(* CODESYS project skyWell.v2.01.project

Project tree, tasks and I/O mapping:
  Device : CODESYS SoftMotion RTE V3, 3S - Smart Software Solutions GmbH, order no. 309015, version 3.5.9.50
    application Application
      libraries: Standard, * (System); VisuDialogs, * (System); SysTime, 3.5.9.0 (System); SysFile, 3.5.9.0 (System); SysStr23, 3.5.8.0 (System); CAA DTUtil Extern, 3.5.10.0 (CAA Technical Workgroup); AC_Persistence, 3.5.10.0 (3S - Smart Software Solutions GmbH); modbus tcp serverAndClient, 1.0.1 (深圳人通长沙研究院); TCP, 3.5.9.50 (3S - Smart Software Solutions GmbH); SysDir, 3.5.8.0 (System); SysTime23, 3.5.2.0 (System); CAA File, 3.5.9.0 (CAA Technical Workgroup)
      task ceilingRail (cyclic, interval t#20ms, priority 1) calls ceilingRailAct
      task healthyData1 (cyclic, interval t#500ms, priority 1) calls tcpUploader
      task VISU_TASK (cyclic, interval 100 ms, priority 31) calls VisuElems.Visu_Prg
      task canSend (cyclic, interval t#20ms, priority 1) calls canTx
      task modbus (cyclic, interval t#20ms, priority 1) calls modbusAct
      task canReceive (cyclic, interval 4 ms, priority 0) calls canRx
      task healthyData2 (cyclic, interval t#10ms, priority 1) calls fileSaver
      rail_ceiling/
        struct_ceiling_rail/
          data type propValveModule_Ti
          data type PropValveTiX
          data type UICell_OilBlock_Ti
        program ceilingRailAct [ST]: initName, statusDisplayTi, initRange, statusPercentCalcTi, cmdDeliverTi, cmdDeliverPlate, cmdDeliverManual
        function cmdExecuteT [ST]
        program positionRecord [ST]
      can/
        structCan/
          data type Can_baseframe
          data type Can_BUS_8Inputs
          data type Can_BUS_8Outputs
          data type Can_Bus_RXMsg_Buff
          data type Can_Bus_TXMsg_Buff
        function CAN_Send_Data_SWMC [ST]
        function swmc_C05_Rx [ST]
        function swmc_C05_Tx [ST]
        function swmc_C06_Tx [ST]
        function swmc_C12_Rx [ST]
        function CAN_Read_Data_SWMC [ST]
        program canTx [ST]
        program canRx [ST]
        function swmc_C06_Rx [ST]
      global variables gImple
      global variables gUI
      global variables gCan
      display/
        Module/
          visualisation OilBlock_PrimButton
          visualisation OilBlock_PrimInfo
          visualisation ModuleX2
          visualisation ModuleX1
          visualisation ModuleX3
          visualisation ModuleX8
          visualisation ModuleX4
          visualisation ModuleX5
          visualisation ModuleDTD
        OrigTi/
          visualisation Ceiling_Rail2
          visualisation Ceiling_Rail1
          visualisation Ceiling_Rail_345
          visualisation Ceiling_Rail6
          visualisation Ceiling_Rail7
          visualisation Ceiling_Rail_12
          visualisation Ceiling_Rail_67
          visualisation Ceiling_Rail_Plate
          visualisation ManualMode
        visualisation Ceiling_Rail
      public_datum/
        yy_station/
          struct_yystation/
            data type YyStation_Cmd
            data type YyStation_Status
            data type YyStation
        oilblock/
          struct/
            data type OilBlockUnit_Base
            data type OilBlockUnit_Status
            data type OilBlockUnit_Cmdx
            data type OilBlockUnit_Status_Loc
            data type OilBlockUnit_Status_PosVal
            data type UICell_OilBlock_Module
            data type UICell_OilBlock_Module_Info
            data type UICell_OilBlock_Module_Button
            data type UICell_OilBlock_Tag
            data type OilBlockUnit_RangeRec
            data type OilBlockUnit_Add
            data type UICell_ManualMode
            data type UICell_OilBlockPlat_Module
        cmdcheck/
          function block checkoilUnit [ST]
          function GetPositionValueOfUnit8 [ST]
          data type cmdStat
          function block checkoilGropisDoneX8 [ST]
          function fGetUnitStat [ST]
          function block percentCalc [ST]
          function block syncUnitCheck [ST]
          function fUICmdDetect [ST]
        datarecord/
          function block datSave [ST]
          function block logSave [ST]
      global variables gModbus
      modbus/
        struct_modbus/
          data type ModbusStructx
          data type Modbus_Commandx
          data type Modbus_Statusx
          data type Modbus_Heartbeatx
          data type Modbus_ActionIndex
        program modbusAct [ST]: initAddrPacket, handleToken, handleCommand1, handleStatus1, executeCmd, getStatus
        function block getObjIndexC [ST]
        function block getObjIndexE [ST]
        function block getObjIndexR [ST]
        function block getColumnStr [ST]
      rail_plate/
        function cmdExecutePlate [ST]
        data type plateCmd
        data type plateStat
      dataUpload/
        function block tcpUpload [ST]: send
        function block findMasterCtrl [ST]
        function block getStateByIdx [ST]
        program tcpUploader [ST]: prepareMetaData
        function block fileSave [ST]: new, close, write, createDir
        program fileSaver [ST]: getData
    SoftMotion General Axis Pool
    EtherCAT_Master : EtherCAT Master, 3S - Smart Software Solutions GmbH, version 3.5.10.0
        settings: NetworkName = '本地连接 2'; NetworkName = "本地连接 2"; SelectNetworkByName = False; SrcAddress1 = 26861; SrcAddress2 = 2752489275
      EK1100_0030_2 : EK1100-0030 EtherCAT Coupler (2A E-Bus, 4kV galv. iso.), Beckhoff Automation GmbH & Co. KG, order no. EK1100-0030, version Revision=16#0011001E
          settings: DC sync0 cycletime = 4000; DC sync1 cycletime = 4000
        EL6751_CANMiniDriver_1 : EL6751 CAN MiniDriver (8 Messages), Beckhoff Automation GmbH, version 3.5.9.0
            settings: DC sync0 cycletime = 4000; DC sync1 cycletime = 4000
            unmapped channels: TxCounter, RxCounter, NoOfTxMessages, TxMsg1_TransactionNumber, TxMsg1_CobId, TxMsg1_Byte1, TxMsg1_Byte2, TxMsg1_Byte3, TxMsg1_Byte4, TxMsg1_Byte5, TxMsg1_Byte6, TxMsg1_Byte7, TxMsg1_Byte8, TxMsg2_TransactionNumber, TxMsg2_CobId, TxMsg2_Byte1, TxMsg2_Byte2, TxMsg2_Byte3, TxMsg2_Byte4, TxMsg2_Byte5, TxMsg2_Byte6, TxMsg2_Byte7, TxMsg2_Byte8, TxMsg3_TransactionNumber, TxMsg3_CobId, TxMsg3_Byte1, TxMsg3_Byte2, TxMsg3_Byte3, TxMsg3_Byte4, TxMsg3_Byte5, TxMsg3_Byte6, TxMsg3_Byte7, TxMsg3_Byte8, TxMsg4_TransactionNumber, TxMsg4_CobId, TxMsg4_Byte1, TxMsg4_Byte2, TxMsg4_Byte3, TxMsg4_Byte4, TxMsg4_Byte5,
              TxMsg4_Byte6, TxMsg4_Byte7, TxMsg4_Byte8, TxMsg5_TransactionNumber, TxMsg5_CobId, TxMsg5_Byte1, TxMsg5_Byte2, TxMsg5_Byte3, TxMsg5_Byte4, TxMsg5_Byte5, TxMsg5_Byte6, TxMsg5_Byte7, TxMsg5_Byte8, TxMsg6_TransactionNumber, TxMsg6_CobId, TxMsg6_Byte1, TxMsg6_Byte2, TxMsg6_Byte3, TxMsg6_Byte4, TxMsg6_Byte5, TxMsg6_Byte6, TxMsg6_Byte7, TxMsg6_Byte8, TxMsg7_TransactionNumber, TxMsg7_CobId, TxMsg7_Byte1, TxMsg7_Byte2, TxMsg7_Byte3, TxMsg7_Byte4, TxMsg7_Byte5, TxMsg7_Byte6, TxMsg7_Byte7, TxMsg7_Byte8, TxMsg8_TransactionNumber, TxMsg8_CobId, TxMsg8_Byte1, TxMsg8_Byte2, TxMsg8_Byte3, TxMsg8_Byte4, TxMsg8_Byte5,
              TxMsg8_Byte6, TxMsg8_Byte7, TxMsg8_Byte8, CAN Control, TxCounter, RxCounter, NoOfRxMessages, TransactionNumber, RxMsg1_CobId, RxMsg1_Byte1, RxMsg1_Byte2, RxMsg1_Byte3, RxMsg1_Byte4, RxMsg1_Byte5, RxMsg1_Byte6, RxMsg1_Byte7, RxMsg1_Byte8, RxMsg2_CobId, RxMsg2_Byte1, RxMsg2_Byte2, RxMsg2_Byte3, RxMsg2_Byte4, RxMsg2_Byte5, RxMsg2_Byte6, RxMsg2_Byte7, RxMsg2_Byte8, RxMsg3_CobId, RxMsg3_Byte1, RxMsg3_Byte2, RxMsg3_Byte3, RxMsg3_Byte4, RxMsg3_Byte5, RxMsg3_Byte6, RxMsg3_Byte7, RxMsg3_Byte8, RxMsg4_CobId, RxMsg4_Byte1, RxMsg4_Byte2, RxMsg4_Byte3, RxMsg4_Byte4,
              RxMsg4_Byte5, RxMsg4_Byte6, RxMsg4_Byte7, RxMsg4_Byte8, RxMsg5_CobId, RxMsg5_Byte1, RxMsg5_Byte2, RxMsg5_Byte3, RxMsg5_Byte4, RxMsg5_Byte5, RxMsg5_Byte6, RxMsg5_Byte7, RxMsg5_Byte8, RxMsg6_CobId, RxMsg6_Byte1, RxMsg6_Byte2, RxMsg6_Byte3, RxMsg6_Byte4, RxMsg6_Byte5, RxMsg6_Byte6, RxMsg6_Byte7, RxMsg6_Byte8, RxMsg7_CobId, RxMsg7_Byte1, RxMsg7_Byte2, RxMsg7_Byte3, RxMsg7_Byte4, RxMsg7_Byte5, RxMsg7_Byte6, RxMsg7_Byte7, RxMsg7_Byte8, RxMsg8_CobId, RxMsg8_Byte1, RxMsg8_Byte2, RxMsg8_Byte3, RxMsg8_Byte4, RxMsg8_Byte5, RxMsg8_Byte6, RxMsg8_Byte7, RxMsg8_Byte8,
              CAN State, Align, RX Error Counter, TX Error Counter
          CANbus
              settings: NetID = 2
      EK1100_0030_1 : EK1100-0030 EtherCAT Coupler (2A E-Bus, 4kV galv. iso.), Beckhoff Automation GmbH & Co. KG, order no. EK1100-0030, version Revision=16#0011001E
          settings: DC sync0 cycletime = 4000; DC sync1 cycletime = 4000
        EL6751_CANMiniDriver : EL6751 CAN MiniDriver (8 Messages), Beckhoff Automation GmbH, version 3.5.9.0
            settings: DC sync0 cycletime = 4000; DC sync1 cycletime = 4000
            unmapped channels: TxCounter, RxCounter, NoOfTxMessages, TxMsg1_TransactionNumber, TxMsg1_CobId, TxMsg1_Byte1, TxMsg1_Byte2, TxMsg1_Byte3, TxMsg1_Byte4, TxMsg1_Byte5, TxMsg1_Byte6, TxMsg1_Byte7, TxMsg1_Byte8, TxMsg2_TransactionNumber, TxMsg2_CobId, TxMsg2_Byte1, TxMsg2_Byte2, TxMsg2_Byte3, TxMsg2_Byte4, TxMsg2_Byte5, TxMsg2_Byte6, TxMsg2_Byte7, TxMsg2_Byte8, TxMsg3_TransactionNumber, TxMsg3_CobId, TxMsg3_Byte1, TxMsg3_Byte2, TxMsg3_Byte3, TxMsg3_Byte4, TxMsg3_Byte5, TxMsg3_Byte6, TxMsg3_Byte7, TxMsg3_Byte8, TxMsg4_TransactionNumber, TxMsg4_CobId, TxMsg4_Byte1, TxMsg4_Byte2, TxMsg4_Byte3, TxMsg4_Byte4, TxMsg4_Byte5,
              TxMsg4_Byte6, TxMsg4_Byte7, TxMsg4_Byte8, TxMsg5_TransactionNumber, TxMsg5_CobId, TxMsg5_Byte1, TxMsg5_Byte2, TxMsg5_Byte3, TxMsg5_Byte4, TxMsg5_Byte5, TxMsg5_Byte6, TxMsg5_Byte7, TxMsg5_Byte8, TxMsg6_TransactionNumber, TxMsg6_CobId, TxMsg6_Byte1, TxMsg6_Byte2, TxMsg6_Byte3, TxMsg6_Byte4, TxMsg6_Byte5, TxMsg6_Byte6, TxMsg6_Byte7, TxMsg6_Byte8, TxMsg7_TransactionNumber, TxMsg7_CobId, TxMsg7_Byte1, TxMsg7_Byte2, TxMsg7_Byte3, TxMsg7_Byte4, TxMsg7_Byte5, TxMsg7_Byte6, TxMsg7_Byte7, TxMsg7_Byte8, TxMsg8_TransactionNumber, TxMsg8_CobId, TxMsg8_Byte1, TxMsg8_Byte2, TxMsg8_Byte3, TxMsg8_Byte4, TxMsg8_Byte5,
              TxMsg8_Byte6, TxMsg8_Byte7, TxMsg8_Byte8, CAN Control, TxCounter, RxCounter, NoOfRxMessages, TransactionNumber, RxMsg1_CobId, RxMsg1_Byte1, RxMsg1_Byte2, RxMsg1_Byte3, RxMsg1_Byte4, RxMsg1_Byte5, RxMsg1_Byte6, RxMsg1_Byte7, RxMsg1_Byte8, RxMsg2_CobId, RxMsg2_Byte1, RxMsg2_Byte2, RxMsg2_Byte3, RxMsg2_Byte4, RxMsg2_Byte5, RxMsg2_Byte6, RxMsg2_Byte7, RxMsg2_Byte8, RxMsg3_CobId, RxMsg3_Byte1, RxMsg3_Byte2, RxMsg3_Byte3, RxMsg3_Byte4, RxMsg3_Byte5, RxMsg3_Byte6, RxMsg3_Byte7, RxMsg3_Byte8, RxMsg4_CobId, RxMsg4_Byte1, RxMsg4_Byte2, RxMsg4_Byte3, RxMsg4_Byte4,
              RxMsg4_Byte5, RxMsg4_Byte6, RxMsg4_Byte7, RxMsg4_Byte8, RxMsg5_CobId, RxMsg5_Byte1, RxMsg5_Byte2, RxMsg5_Byte3, RxMsg5_Byte4, RxMsg5_Byte5, RxMsg5_Byte6, RxMsg5_Byte7, RxMsg5_Byte8, RxMsg6_CobId, RxMsg6_Byte1, RxMsg6_Byte2, RxMsg6_Byte3, RxMsg6_Byte4, RxMsg6_Byte5, RxMsg6_Byte6, RxMsg6_Byte7, RxMsg6_Byte8, RxMsg7_CobId, RxMsg7_Byte1, RxMsg7_Byte2, RxMsg7_Byte3, RxMsg7_Byte4, RxMsg7_Byte5, RxMsg7_Byte6, RxMsg7_Byte7, RxMsg7_Byte8, RxMsg8_CobId, RxMsg8_Byte1, RxMsg8_Byte2, RxMsg8_Byte3, RxMsg8_Byte4, RxMsg8_Byte5, RxMsg8_Byte6, RxMsg8_Byte7, RxMsg8_Byte8,
              CAN State, Align, RX Error Counter, TX Error Counter
          CANbus
              settings: NetID = 1
      EK1100_0030 : EK1100-0030 EtherCAT Coupler (2A E-Bus, 4kV galv. iso.), Beckhoff Automation GmbH & Co. KG, order no. EK1100-0030, version Revision=16#0011001E
          settings: DC sync0 cycletime = 4000; DC sync1 cycletime = 4000
        EL6751_CANMiniDriver_4 : EL6751 CAN MiniDriver (8 Messages), Beckhoff Automation GmbH, version 3.5.9.0
            settings: DC sync0 cycletime = 4000; DC sync1 cycletime = 4000
            unmapped channels: TxCounter, RxCounter, NoOfTxMessages, TxMsg1_TransactionNumber, TxMsg1_CobId, TxMsg1_Byte1, TxMsg1_Byte2, TxMsg1_Byte3, TxMsg1_Byte4, TxMsg1_Byte5, TxMsg1_Byte6, TxMsg1_Byte7, TxMsg1_Byte8, TxMsg2_TransactionNumber, TxMsg2_CobId, TxMsg2_Byte1, TxMsg2_Byte2, TxMsg2_Byte3, TxMsg2_Byte4, TxMsg2_Byte5, TxMsg2_Byte6, TxMsg2_Byte7, TxMsg2_Byte8, TxMsg3_TransactionNumber, TxMsg3_CobId, TxMsg3_Byte1, TxMsg3_Byte2, TxMsg3_Byte3, TxMsg3_Byte4, TxMsg3_Byte5, TxMsg3_Byte6, TxMsg3_Byte7, TxMsg3_Byte8, TxMsg4_TransactionNumber, TxMsg4_CobId, TxMsg4_Byte1, TxMsg4_Byte2, TxMsg4_Byte3, TxMsg4_Byte4, TxMsg4_Byte5,
              TxMsg4_Byte6, TxMsg4_Byte7, TxMsg4_Byte8, TxMsg5_TransactionNumber, TxMsg5_CobId, TxMsg5_Byte1, TxMsg5_Byte2, TxMsg5_Byte3, TxMsg5_Byte4, TxMsg5_Byte5, TxMsg5_Byte6, TxMsg5_Byte7, TxMsg5_Byte8, TxMsg6_TransactionNumber, TxMsg6_CobId, TxMsg6_Byte1, TxMsg6_Byte2, TxMsg6_Byte3, TxMsg6_Byte4, TxMsg6_Byte5, TxMsg6_Byte6, TxMsg6_Byte7, TxMsg6_Byte8, TxMsg7_TransactionNumber, TxMsg7_CobId, TxMsg7_Byte1, TxMsg7_Byte2, TxMsg7_Byte3, TxMsg7_Byte4, TxMsg7_Byte5, TxMsg7_Byte6, TxMsg7_Byte7, TxMsg7_Byte8, TxMsg8_TransactionNumber, TxMsg8_CobId, TxMsg8_Byte1, TxMsg8_Byte2, TxMsg8_Byte3, TxMsg8_Byte4, TxMsg8_Byte5,
              TxMsg8_Byte6, TxMsg8_Byte7, TxMsg8_Byte8, CAN Control, TxCounter, RxCounter, NoOfRxMessages, TransactionNumber, RxMsg1_CobId, RxMsg1_Byte1, RxMsg1_Byte2, RxMsg1_Byte3, RxMsg1_Byte4, RxMsg1_Byte5, RxMsg1_Byte6, RxMsg1_Byte7, RxMsg1_Byte8, RxMsg2_CobId, RxMsg2_Byte1, RxMsg2_Byte2, RxMsg2_Byte3, RxMsg2_Byte4, RxMsg2_Byte5, RxMsg2_Byte6, RxMsg2_Byte7, RxMsg2_Byte8, RxMsg3_CobId, RxMsg3_Byte1, RxMsg3_Byte2, RxMsg3_Byte3, RxMsg3_Byte4, RxMsg3_Byte5, RxMsg3_Byte6, RxMsg3_Byte7, RxMsg3_Byte8, RxMsg4_CobId, RxMsg4_Byte1, RxMsg4_Byte2, RxMsg4_Byte3, RxMsg4_Byte4,
              RxMsg4_Byte5, RxMsg4_Byte6, RxMsg4_Byte7, RxMsg4_Byte8, RxMsg5_CobId, RxMsg5_Byte1, RxMsg5_Byte2, RxMsg5_Byte3, RxMsg5_Byte4, RxMsg5_Byte5, RxMsg5_Byte6, RxMsg5_Byte7, RxMsg5_Byte8, RxMsg6_CobId, RxMsg6_Byte1, RxMsg6_Byte2, RxMsg6_Byte3, RxMsg6_Byte4, RxMsg6_Byte5, RxMsg6_Byte6, RxMsg6_Byte7, RxMsg6_Byte8, RxMsg7_CobId, RxMsg7_Byte1, RxMsg7_Byte2, RxMsg7_Byte3, RxMsg7_Byte4, RxMsg7_Byte5, RxMsg7_Byte6, RxMsg7_Byte7, RxMsg7_Byte8, RxMsg8_CobId, RxMsg8_Byte1, RxMsg8_Byte2, RxMsg8_Byte3, RxMsg8_Byte4, RxMsg8_Byte5, RxMsg8_Byte6, RxMsg8_Byte7, RxMsg8_Byte8,
              CAN State, Align, RX Error Counter, TX Error Counter
          CANbus
  libraries: VisuSymbols, 3.5.10.0 (System)
  text list GlobalTextList
*)

// Device/Application/public_datum/yy_station/struct_yystation/YyStation_Cmd
TYPE YyStation_Cmd :
STRUCT
	InverterFan_Ctrl  		:BOOL;   //变频风机控制 0x400-1.0
	OilPumpFan_Ctrl   		:BOOL;   //油泵风机控制 0x400-1.1
	//------以下变量暂未使用,取自水平库-----------------------------------
	OilPumpMotor_Ctrl 		:BOOL;   //油泵电机控制
	OilPumpMotor_PN_Ctrl 	:BOOL;   //油泵电机正反转控制
	HL_Mode_Ctrl 			:BOOL;   //高低速模式
	KEEP_Mode_Ctrl          :BOOL;   //恒速模式
	Energy_Swith			:BOOL;   //储能控制
	Oil_Pre_Val             :WORD;   //油压控制
END_STRUCT
END_TYPE

// Device/Application/public_datum/yy_station/struct_yystation/YyStation_Status
TYPE YyStation_Status :
STRUCT

	pressureStatus					: REAL;		//压力开关S1|0x300-Byt1~2
	temperatureStatus				: REAL;		//温度开关S14|0x300-Byt3~4
	yeweiStatus						: BOOL;		//液位开关S15|0x300-Byt5~6

	FrequencyConversion_Fault 		: BOOL;			//变频故障|0x300-7.0
	FrequencyConversion_Run 		: BOOL;			//变频运行|0x300-7.1
	HydraulicStation_Power			: BOOL;			//液压站上电-状态|0x300-7.2
	Control_Power					: BOOL;			//控制总电源上电状态|0x300-7.3
	InverterFan_Run 				: BOOL;			//变频风机运行状态|0x300-7.4
	OilPumpFan						: BOOL;			//冷却油泵状态|0x300-7.5
	OilPumpM_Fault 					: BOOL;			//油泵电机故障状态|0x300-7.6
	InverterFan_Fault 				: BOOL;			//变频风机故障|0x300-7.7
	
	//地轨部分压力传感器
	pressureV2						: REAL;			//压力传感器S2P|0x316-Byt1~2
	pressureV3						: REAL;			//压力传感器S3P|0x316-Byt3~4
	pressureV4						: REAL;			//压力传感器S4P|0x326-Byt1~2
	pressureV5						: REAL;			//压力传感器S5P|0x326-Byt3~4
	//天轨部分压力传感器
	pressureV8						: REAL;			//压力传感器S8P|0x356-Byt1~2
	pressureV9						: REAL;			//压力传感器S9P|0x356-Byt3~4
	pressureV10						: REAL;			//压力传感器S10P|0x366-Byt1~2
	pressureV11						: REAL;			//压力传感器S11P|0x366-Byt3~4
	
	arrSL							:ARRAY[1..2] OF BOOL;			//限位开关状态

	

END_STRUCT
END_TYPE

// Device/Application/public_datum/yy_station/struct_yystation/YyStation
TYPE YyStation :
STRUCT
	Cmd		:YyStation_Cmd;		//液压站指令
	Status	:YyStation_Status;	//液压站状态
	
END_STRUCT
END_TYPE

// Device/Application/can/structCan/Can_baseframe
TYPE Can_baseframe :
STRUCT
	id		: UINT;
	data	: ARRAY[1..8] OF BYTE;
END_STRUCT
END_TYPE

// Device/Application/can/structCan/Can_BUS_8Inputs
TYPE Can_BUS_8Inputs :          //输入缓存结构 EL6751-8Message_IN
STRUCT
	TxCounter			: UINT;
	RxCounter			: UINT;
	NoOfRxMessages 	 	: UINT;
	TransactionNumber	: UINT;
	RXMsg				: ARRAY[1..8] OF Can_Bus_RXMsg_Buff;
	CAN_State			: UINT;
	Align				: UINT;
	RX_Error_Cnt		: BYTE;
	TX_Error_Cnt		: BYTE;
END_STRUCT
END_TYPE

// Device/Application/can/structCan/Can_BUS_8Outputs
TYPE Can_BUS_8Outputs :		//输出缓存结构 EL6751-8Message_OUT
STRUCT
	TxCounter		: UINT;
	RxCounter		: UINT;
	NoOfTxMessages 	: UINT;
	TXMsg			: ARRAY[1..8] OF Can_Bus_TXMsg_Buff;
	CAN_Control		: UINT;
END_STRUCT
END_TYPE

// Device/Application/can/structCan/Can_Bus_RXMsg_Buff
TYPE Can_Bus_RXMsg_Buff:
STRUCT
	RxMsg_CobId		: UINT;
	RxMsg_Byte  	: ARRAY[1..8] OF BYTE;
END_STRUCT
END_TYPE

// Device/Application/can/structCan/Can_Bus_TXMsg_Buff
TYPE Can_Bus_TXMsg_Buff :
STRUCT
	TxMsg_TransactionNumber		: UINT;
	TxMsg_CobId					: UINT;
	TxMsg_Byte  				: ARRAY[1..8] OF BYTE;
END_STRUCT
END_TYPE

// Device/Application/public_datum/oilblock/struct/OilBlockUnit_Base
TYPE OilBlockUnit_Base :
STRUCT
	cmd		:OilBlockUnit_Cmd;				//发送油缸指令
	status	:OilBlockUnit_Status;			//油缸状态
	cnt     :UINT;			  				//超时计数

END_STRUCT
END_TYPE

// Device/Application/public_datum/oilblock/struct/OilBlockUnit_Status
TYPE OilBlockUnit_Status :
STRUCT
	
	posVal			:OilBlockUnit_Status_PosVal;	//传感器位置值
	locStat			:OilBlockUnit_Status_Loc;		//位置状态（枚举类单个插销状态）
	
END_STRUCT
END_TYPE

// Device/Application/public_datum/oilblock/struct/OilBlockUnit_Cmdx
TYPE OilBlockUnit_Cmdx :
STRUCT
	bE_Open		:BOOL;				//插销伸出指令
	bR_Open 	:BOOL;				//插销缩回指令
	
	eStat		:cmdStat;			//单开关阀总状态参数


END_STRUCT
END_TYPE

// Device/Application/public_datum/oilblock/struct/OilBlockUnit_Status_Loc
{attribute 'qualified_only'}
{attribute 'strict'}
TYPE OilBlockUnit_Status_Loc :
(
	eUnknow  		:=  0,   

	eExtended 		:= 10,	//伸出完成
	eRetracted  	:= 20,	//缩回完成
	eRunning		:= 30,	//运行中
	
	eErr  			:= 90   //错误
);
END_TYPE

// Device/Application/public_datum/oilblock/struct/OilBlockUnit_Status_PosVal
TYPE OilBlockUnit_Status_PosVal :
STRUCT
	Extend 		:REAL;    //伸出位置
	Retract   	:REAL;    //收回位置
	Current 	:REAL;    //当前位置
END_STRUCT
END_TYPE

// Device/Application/public_datum/oilblock/struct/UICell_OilBlock_Module
TYPE UICell_OilBlock_Module :
STRUCT
	
	bPVD_enable			:BOOL;			//比例阀使能
	rPVDPercent			:REAL;			//比例阀百分比

	sColumn				:ARRAY[1..8] OF UICell_OilBlock_Module_Button;	//最小控制插销组按钮	
	sNum				:ARRAY[1..24] OF UICell_OilBlock_Module_Info;	//插销缸信息

END_STRUCT
END_TYPE

// Device/Application/public_datum/oilblock/struct/UICell_OilBlock_Module_Info
TYPE UICell_OilBlock_Module_Info :
STRUCT
	strName			:STRING;	//编号
	rPosition		:REAL;		//传感器位移值
	rPercent		:REAL;		//伸出百分比
END_STRUCT
END_TYPE

// Device/Application/public_datum/oilblock/struct/UICell_OilBlock_Module_Button
TYPE UICell_OilBlock_Module_Button :
STRUCT
	bExtend			: BOOL;			//伸出按钮
	bRetract		: BOOL;			//缩回按钮
	bStop			: BOOL;			//停止按钮
	
	cmdLast			:cmdStat;
	//cmdNew			:cmdStat;
END_STRUCT
END_TYPE

// Device/Application/public_datum/oilblock/struct/UICell_OilBlock_Tag
TYPE UICell_OilBlock_Tag :
STRUCT
	strName				:ARRAY[1..7,1..24] OF STRING;
	
END_STRUCT
END_TYPE

// Device/Application/public_datum/oilblock/struct/OilBlockUnit_RangeRec
TYPE OilBlockUnit_RangeRec :
STRUCT
	rRetract				:ARRAY[1..7,1..24] OF REAL;//标定的伸出值
	rExtend					:ARRAY[1..7,1..24] OF REAL;//标定的缩回值
	
	numHead					:ARRAY[1..7,1..7] OF INT;
	numTail					:ARRAY[1..7,1..7] OF INT;
	numInColumn				:ARRAY[1..7,1..7] OF INT;//对应序号内的插销数量
	
END_STRUCT
END_TYPE

// Device/Application/rail_ceiling/struct_ceiling_rail/propValveModule_Ti
TYPE propValveModule_Ti :
STRUCT
	arrPV				:ARRAY[1..7] OF PropValveTiX;		//直线部分
	arrAddtion			:ARRAY[1..2] OF OilBlockUnit_Add;	//附加部分

END_STRUCT
END_TYPE

// Device/Application/rail_ceiling/struct_ceiling_rail/PropValveTiX
TYPE PropValveTiX :
STRUCT
	
	percenVal			:WORD;  								//比例阀
	
	sColumn				:ARRAY[1..7]  OF OilBlockUnit_Cmdx;		//发送油缸指令
	iCntErr    			:ARRAY[1..7]  OF UINT;			  		//超时计数
	sNum				:ARRAY[1..24] OF OilBlockUnit_Status;	//油缸状态
	
END_STRUCT
END_TYPE

// Device/Application/rail_ceiling/struct_ceiling_rail/UICell_OilBlock_Ti
TYPE UICell_OilBlock_Ti :
STRUCT
	
	arrPV		:ARRAY[1..7] OF UICell_OilBlock_Module;			//插销缸模块
	arrPlate	:ARRAY[1..2] OF UICell_OilBlockPlat_Module;		//挡板模块
END_STRUCT
END_TYPE

// Device/Application/public_datum/oilblock/struct/OilBlockUnit_Add
TYPE OilBlockUnit_Add :
STRUCT
	
	sPlateCtrl		:plateCmd;		//挡板控制
	sPlateStatus	:plateStat;		//挡板状态
	

	
END_STRUCT
END_TYPE

// Device/Application/public_datum/oilblock/struct/UICell_ManualMode
TYPE UICell_ManualMode :
STRUCT
	bCmdReset				:BOOL;//指令复位手动模式->1
	bDteEnable				:BOOL;//比例阀门使能手动->1
END_STRUCT
END_TYPE

// Device/Application/public_datum/cmdcheck/cmdStat
{attribute 'qualified_only'}
{attribute 'strict'}
TYPE cmdStat :
(
	eNormal 	 	:= 0,   //正常态
	eRun			:= 1,	//运行态
	eFree 	 		:= 2,   //空闲态

	
	
	cExtend  		:= 10,	//伸出指令
	Extend_Run		:= 11,  //伸出运行状态
	Extend_Done		:= 12,  //伸出完成状态
	
	cRetract 		:= 20,  //收回指令
	Retract_Run 	:= 21,  //收回运行
	Retract_Done	:= 22,	//收回完成状态
	
	cStop			:= 40,	//停止指令
	
	Stop_Done		:= 42,	//停止完成状态
	
	
	Unknow			:= 90,	//未知
	eError 			:= 99   //错误状态
);
END_TYPE

// Device/Application/modbus/struct_modbus/ModbusStructx
TYPE ModbusStructx :
STRUCT
	
	sToken			:Modbus_ActionIndex;	//编号
	sCmd			:Modbus_Commandx;		//指令
	sStatus			:Modbus_Statusx;		//状态
	//sHeartbeat	:Modbus_Heartbeatx;			//心跳
END_STRUCT
END_TYPE

// Device/Application/modbus/struct_modbus/Modbus_Commandx
TYPE Modbus_Commandx :
STRUCT
	wStartAddr		:WORD;					//解析起始地址/10
	wAmount			:WORD;					//解析数量/48
	arrDat			:ARRAY[10..57] OF WORD;	//指令数据
	
	wRotplatNew		:WORD;					//转台数据帧：1WORD
	wRotplatLast	:WORD;	
	arrNew		:ARRAY [10..15,0..15] OF BOOL;
	arrLast		:ARRAY [10..15,0..15] OF BOOL;
END_STRUCT
END_TYPE

// Device/Application/modbus/struct_modbus/Modbus_Statusx
TYPE Modbus_Statusx :
STRUCT
	wStartAddr		:WORD;						//解析起始地址/110
	wAmount			:WORD;						//解析数量/205-110+1
	arrDat			:ARRAY[110..205] OF WORD;	//位置数据

	//arrRot		:ARRAY[241..244] OF WORD;	//天轨转台位置数据
	//newarrDat		:ARRAY[110..167] OF WORD;	//位置数据
	//arrTemp		:ARRAY[1..7,1..7] OF USINT;
END_STRUCT
END_TYPE

// Device/Application/modbus/struct_modbus/Modbus_Heartbeatx
TYPE Modbus_Heartbeatx :
STRUCT
	wStartAddr		:WORD;	//解析起始地址
	wAmount			:WORD;	//解析数量
	iHeartNum		:WORD;	//心跳数
END_STRUCT
END_TYPE

// Device/Application/modbus/struct_modbus/Modbus_ActionIndex
TYPE Modbus_ActionIndex :
STRUCT
	wStartAddr		:WORD;	//解析起始地址/42
	wAmount			:WORD;	//解析数量/1
	iNo				:WORD;	//指令序号，新指令会加1区分旧指令
	iLast			:WORD;
	iNew			:WORD;
END_STRUCT
END_TYPE

// Device/Application/public_datum/oilblock/struct/UICell_OilBlockPlat_Module
TYPE UICell_OilBlockPlat_Module :
STRUCT
	sCmd				: UICell_OilBlock_Module_Button;	//转台界面指令按钮
	sInfo				: UICell_OilBlock_Module_Info;		//转台界面信息
END_STRUCT
END_TYPE

// Device/Application/rail_plate/plateCmd
TYPE plateCmd :
STRUCT
	bExtend		:BOOL;	//挡板伸出
	bRetract	:BOOL;	//挡板到位
END_STRUCT
END_TYPE

// Device/Application/rail_plate/plateStat
TYPE plateStat :
STRUCT


	sSensor				:OilBlockUnit_Status_PosVal;		//传感器位移值
	eStat				:cmdStat;							//转台枚举类状态	
	iCnt				:UINT;								//计数器
END_STRUCT
END_TYPE

// Device/Application/gImple
{attribute 'qualified_only'}
VAR_GLOBAL
	
	//液压站
	//hydraPresStation	:YyStation;

	//天轨
	PV_GroupTi			:propValveModule_Ti;	//天轨控制结构
	TiG_InitPacket		:OilBlockUnit_RangeRec;	//天轨初始化信息

END_VAR

// Device/Application/gUI
{attribute 'qualified_only'}
VAR_GLOBAL
	
	sManualMode					:UICell_ManualMode;

	//天轨比例阀单元
	TiG							:UICell_OilBlock_Ti;
	TiG_NameInit				:UICell_OilBlock_Tag;
	
	
END_VAR

// Device/Application/gCan
{attribute 'qualified_only'}
VAR_GLOBAL
	//SWMC		
	
	C6TxMsg				AT%QW00:Can_BUS_8Outputs;	
	C6RxMsg				AT%IW00:Can_BUS_8Inputs;
	C6RxCounter			 	   : UINT;
	
	C12TxMsg			AT%QW52:Can_BUS_8Outputs;	
	C12RxMsg			AT%IW47:Can_BUS_8Inputs;
	C12RxCounter			   : UINT;

	C5TxMsg				AT%QW104:Can_BUS_8Outputs;	
	C5RxMsg				AT%IW94:Can_BUS_8Inputs;
	C5RxCounter				   : UINT;

	
END_VAR

// Device/Application/gModbus
{attribute 'qualified_only'}
VAR_GLOBAL CONSTANT
	g_modbusDataSizeMax	:  UINT:=65535; // 从机保持寄存器数量
END_VAR

VAR_GLOBAL
	master			:ModbusStructx;
	arrBufferDat	:ARRAY[0..g_modbusDataSizeMax] OF WORD;	//输入寄存器数据区
END_VAR

// Device/Application/rail_ceiling/ceilingRailAct
PROGRAM ceilingRailAct
VAR
	bInitialize		:BOOL:=TRUE;
	bPropValveIsOn	:BOOL;
	iVT				:INT;
	iVT1			:INT;
	iTemp			:INT;
	rTemp			:REAL;
	fbPercenOut		:percentCalc;
END_VAR
VAR CONSTANT
	aNo		:ARRAY [1..7] OF INT :=[6, 5,1,1,1,5, 7];		//每个比例阀下开关阀的数量(天轨):arrMappingRealNumTiG
	aOil	:ARRAY [1..7] OF INT :=[9,11,8,8,8,8,23];		
END_VAR


IF bInitialize THEN								//初始化
	ceilingRailAct.initName();
	ceilingRailAct.initRange();
	FOR iTemp:=1 TO 7 DO
		gUI.TiG.arrPV[iTemp].rPVDPercent:=80;	//打开对应比例阀，开度设定为80%
	END_FOR
	bInitialize:=FALSE;
END_IF

ceilingRailAct.statusDisplayTi();				//状态显示

IF gUI.sManualMode.bCmdReset THEN
	ceilingRailAct.cmdDeliverManual();			//手动复位指令模式
ELSE
	ceilingRailAct.cmdDeliverTi();				//带自动复位的指令发送模式-插销部分
	ceilingRailAct.cmdDeliverPlate();			//挡板
END_IF

IF gUI.sManualMode.bDteEnable THEN
	//iTemp:=1;
ELSE
	//打开比例阀：有指令打开，无指令关闭->通过检测界面按钮实现
	bPropValveIsOn:=fUICmdDetect(ADR(gUI.TiG));
	IF bPropValveIsOn THEN
		FOR iTemp:=1 TO 7 DO
			gUI.TiG.arrPV[iTemp].bPVD_enable:=TRUE;
		END_FOR
	ELSE
		FOR iTemp:=1 TO 7 DO
			gUI.TiG.arrPV[iTemp].bPVD_enable:=FALSE;
		END_FOR
	END_IF
END_IF

ACTION initName:
gUI.TiG_NameInit.strName[1,1]:='E28L1';
gUI.TiG_NameInit.strName[1,2]:='E28L2';
gUI.TiG_NameInit.strName[1,3]:='E29L';
gUI.TiG_NameInit.strName[1,4]:='E30L';
gUI.TiG_NameInit.strName[1,5]:='E00L';
gUI.TiG_NameInit.strName[1,6]:='E29Q';
gUI.TiG_NameInit.strName[1,7]:='E30Q';
gUI.TiG_NameInit.strName[1,8]:='E28Q';
gUI.TiG_NameInit.strName[1,9]:='E01L';

gUI.TiG_NameInit.strName[2,1]:='E02L';
gUI.TiG_NameInit.strName[2,2]:='E03L';
gUI.TiG_NameInit.strName[2,3]:='E04L';
gUI.TiG_NameInit.strName[2,4]:='E05L';
gUI.TiG_NameInit.strName[2,5]:='E06L';
gUI.TiG_NameInit.strName[2,6]:='E07L';
gUI.TiG_NameInit.strName[2,7]:='E08L';
gUI.TiG_NameInit.strName[2,8]:='E09L';
gUI.TiG_NameInit.strName[2,9]:='E10L';
gUI.TiG_NameInit.strName[2,10]:='E11L';
gUI.TiG_NameInit.strName[2,11]:='E12L';

gUI.TiG_NameInit.strName[3,1]:='E01Q1';
gUI.TiG_NameInit.strName[3,2]:='E01Q2';
gUI.TiG_NameInit.strName[3,3]:='E02Q1';
gUI.TiG_NameInit.strName[3,4]:='E02Q2';
gUI.TiG_NameInit.strName[3,5]:='E03Q1';
gUI.TiG_NameInit.strName[3,6]:='E03Q2';
gUI.TiG_NameInit.strName[3,7]:='E04Q1';
gUI.TiG_NameInit.strName[3,8]:='E04Q2';
gUI.TiG_NameInit.strName[4,1]:='E05Q1';
gUI.TiG_NameInit.strName[4,2]:='E05Q2';
gUI.TiG_NameInit.strName[4,3]:='E06Q1';
gUI.TiG_NameInit.strName[4,4]:='E06Q2';
gUI.TiG_NameInit.strName[4,5]:='E07Q1';
gUI.TiG_NameInit.strName[4,6]:='E07Q2';
gUI.TiG_NameInit.strName[4,7]:='E08Q1';
gUI.TiG_NameInit.strName[4,8]:='E08Q2';
gUI.TiG_NameInit.strName[5,1]:='E09Q1';
gUI.TiG_NameInit.strName[5,2]:='E09Q2';
gUI.TiG_NameInit.strName[5,3]:='E10Q1';
gUI.TiG_NameInit.strName[5,4]:='E10Q2';
gUI.TiG_NameInit.strName[5,5]:='E11Q1';
gUI.TiG_NameInit.strName[5,6]:='E11Q2';
gUI.TiG_NameInit.strName[5,7]:='E12Q1';
gUI.TiG_NameInit.strName[5,8]:='E12Q2';

gUI.TiG_NameInit.strName[6,1]:='E13Q';
gUI.TiG_NameInit.strName[6,2]:='E14Q';
gUI.TiG_NameInit.strName[6,3]:='E15Q';
gUI.TiG_NameInit.strName[6,4]:='E14L';
gUI.TiG_NameInit.strName[6,5]:='E15L';
gUI.TiG_NameInit.strName[6,6]:='E13L';
gUI.TiG_NameInit.strName[6,7]:='E16L1';
gUI.TiG_NameInit.strName[6,8]:='E16L2';

gUI.TiG_NameInit.strName[7,1]:='E18L';
gUI.TiG_NameInit.strName[7,2]:='E19L';
gUI.TiG_NameInit.strName[7,3]:='E20L';
gUI.TiG_NameInit.strName[7,4]:='E21L';
gUI.TiG_NameInit.strName[7,5]:='E22L';
gUI.TiG_NameInit.strName[7,6]:='E23L';
gUI.TiG_NameInit.strName[7,7]:='E24L';
gUI.TiG_NameInit.strName[7,8]:='E25L';
gUI.TiG_NameInit.strName[7,9]:='E26L';
gUI.TiG_NameInit.strName[7,10]:='E17Q';
gUI.TiG_NameInit.strName[7,11]:='E18Q';
gUI.TiG_NameInit.strName[7,12]:='E19Q';
gUI.TiG_NameInit.strName[7,13]:='E20Q';
gUI.TiG_NameInit.strName[7,14]:='E21Q';
gUI.TiG_NameInit.strName[7,15]:='E22Q';
gUI.TiG_NameInit.strName[7,16]:='E23Q';
gUI.TiG_NameInit.strName[7,17]:='E24Q';
gUI.TiG_NameInit.strName[7,18]:='E25Q';
gUI.TiG_NameInit.strName[7,19]:='E26Q';
gUI.TiG_NameInit.strName[7,20]:='E17L1';
gUI.TiG_NameInit.strName[7,21]:='E17L2';
gUI.TiG_NameInit.strName[7,22]:='E27L1';
gUI.TiG_NameInit.strName[7,23]:='E27L2';


FOR iVT:=1 TO 7 DO
	FOR iVT1:=1 TO aOil[iVT] DO
		gUI.TiG.arrPV[iVT].sNum[iVT1].strName:=gUI.TiG_NameInit.strName[iVT,iVT1];

	END_FOR
END_FOR

gUI.TiG.arrPlate[1].sInfo.strName:='Plate1';
gUI.TiG.arrPlate[2].sInfo.strName:='Plate2';
END_ACTION

ACTION statusDisplayTi:

//按比例阀顺序：每油缸位置显示--行程百分比计算

FOR iVT:=1 TO 7 DO
	FOR iVT1:=1 TO aOil[iVT] DO
		gUI.TiG.arrPV[iVT].sNum[iVT1].rPosition:=gImple.PV_GroupTi.arrPV[iVT].sNum[iVT1].posVal.Current;
		gUI.TiG.arrPV[iVT].sNum[iVT1].rPercent:=statusPercentCalcTi(ADR(gImple.PV_GroupTi),iVT,iVT1);
	END_FOR
END_FOR

gUI.TiG.arrPlate[1].sInfo.rPosition:=gImple.PV_GroupTi.arrAddtion[1].sPlateStatus.sSensor.Current;
fbPercenOut(rInput:=gImple.PV_GroupTi.arrAddtion[1].sPlateStatus.sSensor.Current,
			rExtend:=gImple.PV_GroupTi.arrAddtion[1].sPlateStatus.sSensor.Extend,
			rRetract:=gImple.PV_GroupTi.arrAddtion[1].sPlateStatus.sSensor.Retract,
			rOut=>rTemp);
gUI.TiG.arrPlate[1].sInfo.rPercent:=rTemp;			


gUI.TiG.arrPlate[2].sInfo.rPosition:=gImple.PV_GroupTi.arrAddtion[2].sPlateStatus.sSensor.Current;
fbPercenOut(rInput:=gImple.PV_GroupTi.arrAddtion[2].sPlateStatus.sSensor.Current,
			rExtend:=gImple.PV_GroupTi.arrAddtion[2].sPlateStatus.sSensor.Extend,
			rRetract:=gImple.PV_GroupTi.arrAddtion[2].sPlateStatus.sSensor.Retract,
			rOut=>rTemp);
gUI.TiG.arrPlate[2].sInfo.rPercent:=rTemp;	

(*
//比例阀DTE1
FOR iVT	:=1 TO 9 DO
	gUI.TiG.arrPV[1].sNum[iVT].rPosition:=gImple.PV_GroupTi.arrPV[1].sNum[iVT].posVal.Current;
	gUI.TiG.arrPV[1].sNum[iVT].rPercent:=statusPercentCalcTi(ADR(gImple.PV_GroupTi),1,iVT);
	
END_FOR

//比例阀DTE2
FOR iVT	:=1 TO 11 DO
	gUI.TiG.arrPV[2].sNum[iVT].rPosition:=gImple.PV_GroupTi.arrPV[2].sNum[iVT].posVal.Current;
	gUI.TiG.arrPV[2].sNum[iVT].rPercent:=statusPercentCalcTi(ADR(gImple.PV_GroupTi),2,iVT);

END_FOR

//比例阀DTE345
FOR iVT	:=1 TO 8 DO
	gUI.TiG.arrPV[3].sNum[iVT].rPosition:=gImple.PV_GroupTi.arrPV[3].sNum[iVT].posVal.Current;
	gUI.TiG.arrPV[4].sNum[iVT].rPosition:=gImple.PV_GroupTi.arrPV[4].sNum[iVT].posVal.Current;
	gUI.TiG.arrPV[5].sNum[iVT].rPosition:=gImple.PV_GroupTi.arrPV[5].sNum[iVT].posVal.Current;
		
	gUI.TiG.arrPV[3].sNum[iVT].rPercent:=statusPercentCalcTi(ADR(gImple.PV_GroupTi),3,iVT);
	gUI.TiG.arrPV[4].sNum[iVT].rPercent:=statusPercentCalcTi(ADR(gImple.PV_GroupTi),4,iVT);
	gUI.TiG.arrPV[5].sNum[iVT].rPercent:=statusPercentCalcTi(ADR(gImple.PV_GroupTi),5,iVT);

END_FOR

//比例阀DTE6
FOR iVT	:=1 TO 8 DO
	gUI.TiG.arrPV[6].sNum[iVT].rPosition:=gImple.PV_GroupTi.arrPV[6].sNum[iVT].posVal.Current;
	gUI.TiG.arrPV[6].sNum[iVT].rPercent:=statusPercentCalcTi(ADR(gImple.PV_GroupTi),6,iVT);
END_FOR

//比例阀DTE7
FOR iVT	:=1 TO 23 DO
	gUI.TiG.arrPV[7].sNum[iVT].rPosition:=gImple.PV_GroupTi.arrPV[7].sNum[iVT].posVal.Current;
	gUI.TiG.arrPV[7].sNum[iVT].rPercent:=statusPercentCalcTi(ADR(gImple.PV_GroupTi),7,iVT);
END_FOR
*)
END_ACTION

ACTION initRange:
//标定
gImple.TiG_InitPacket.rRetract[1,1]:=	23.8	;	gImple.TiG_InitPacket.rExtend[1,1]:=	72.6	-25;	//E28L1
gImple.TiG_InitPacket.rRetract[1,2]:=	23.7	;	gImple.TiG_InitPacket.rExtend[1,2]:=	72.3	-25;	//E28L2
gImple.TiG_InitPacket.rRetract[1,3]:=	33.3	;	gImple.TiG_InitPacket.rExtend[1,3]:=	97.0	-30;	//E29L
	//gImple.TiG_InitPacket.rRetract[1,4]:=	34.3	;	gImple.TiG_InitPacket.rExtend[1,4]:=	98.1	-30;	//E30L
gImple.TiG_InitPacket.rRetract[1,4]:=	45.0	;	gImple.TiG_InitPacket.rExtend[1,4]:=	108.7	-30;	//E30L
gImple.TiG_InitPacket.rRetract[1,5]:=	32.6	;	gImple.TiG_InitPacket.rExtend[1,5]:=	210.1	-30;	//E00L //218.1;	
gImple.TiG_InitPacket.rRetract[1,6]:=	33.0	;	gImple.TiG_InitPacket.rExtend[1,6]:=	81.7	-20;	//E29Q
gImple.TiG_InitPacket.rRetract[1,7]:=	35.2	;	gImple.TiG_InitPacket.rExtend[1,7]:=	83.7	-20;	//E30Q
gImple.TiG_InitPacket.rRetract[1,8]:=	32.5	;	gImple.TiG_InitPacket.rExtend[1,8]:=	81.1	-20;	//E28Q
gImple.TiG_InitPacket.rRetract[1,9]:=	34.9	;	gImple.TiG_InitPacket.rExtend[1,9]:=	98.5	-30;	//E01L
						
gImple.TiG_InitPacket.rRetract[2,1]:=	34.4	;	gImple.TiG_InitPacket.rExtend[2,1]:=	98.0	-30;	//E02L
gImple.TiG_InitPacket.rRetract[2,2]:=	35.2	;	gImple.TiG_InitPacket.rExtend[2,2]:=	99.0	-30;	//E03L
gImple.TiG_InitPacket.rRetract[2,3]:=	35.1	;	gImple.TiG_InitPacket.rExtend[2,3]:=	98.7	-30;	//E04L
gImple.TiG_InitPacket.rRetract[2,4]:=	32.1	;	gImple.TiG_InitPacket.rExtend[2,4]:=	95.8	-30;	//E05L
gImple.TiG_InitPacket.rRetract[2,5]:=	32.3	;	gImple.TiG_InitPacket.rExtend[2,5]:=	95.9	-30;	//E06L
gImple.TiG_InitPacket.rRetract[2,6]:=	33.5	;	gImple.TiG_InitPacket.rExtend[2,6]:=	97.1	-30;	//E07L
gImple.TiG_InitPacket.rRetract[2,7]:=	32.7	;	gImple.TiG_InitPacket.rExtend[2,7]:=	96.3	-30;	//E08L
gImple.TiG_InitPacket.rRetract[2,8]:=	32.4	;	gImple.TiG_InitPacket.rExtend[2,8]:=	96.4	-30;	//E09L
gImple.TiG_InitPacket.rRetract[2,9]:=	33.6	;	gImple.TiG_InitPacket.rExtend[2,9]:=	96.3	-30;	//E10L
gImple.TiG_InitPacket.rRetract[2,10]:=	33.7	;	gImple.TiG_InitPacket.rExtend[2,10]:=	97.0	-30;	//E11L
gImple.TiG_InitPacket.rRetract[2,11]:=	34.8	;	gImple.TiG_InitPacket.rExtend[2,11]:=	97.0	-30;	//E12L
						
gImple.TiG_InitPacket.rRetract[3,1]:=	37.3	;	gImple.TiG_InitPacket.rExtend[3,1]:=	85.9	-20;	//E01Q1
gImple.TiG_InitPacket.rRetract[3,2]:=	35.2	;	gImple.TiG_InitPacket.rExtend[3,2]:=	83.6	-20;	//E01Q2
gImple.TiG_InitPacket.rRetract[3,3]:=	35.3	;	gImple.TiG_InitPacket.rExtend[3,3]:=	83.9	-20;	//E02Q1
gImple.TiG_InitPacket.rRetract[3,4]:=	34.7	;	gImple.TiG_InitPacket.rExtend[3,4]:=	83.3	-20;	//E02Q2
gImple.TiG_InitPacket.rRetract[3,5]:=	34.6	;	gImple.TiG_InitPacket.rExtend[3,5]:=	83.6	-20;	//E03Q1
gImple.TiG_InitPacket.rRetract[3,6]:=	35.9	;	gImple.TiG_InitPacket.rExtend[3,6]:=	84.3	-20;	//E03Q2
gImple.TiG_InitPacket.rRetract[3,7]:=	35.4	;	gImple.TiG_InitPacket.rExtend[3,7]:=	84.0	-20;	//E04Q1
gImple.TiG_InitPacket.rRetract[3,8]:=	35.9	;	gImple.TiG_InitPacket.rExtend[3,8]:=	84.4	-20;	//E04Q2
gImple.TiG_InitPacket.rRetract[4,1]:=	32.5	;	gImple.TiG_InitPacket.rExtend[4,1]:=	81.1	-20;	//E05Q1
gImple.TiG_InitPacket.rRetract[4,2]:=	31.8	;	gImple.TiG_InitPacket.rExtend[4,2]:=	80.3	-20;	//E05Q2
gImple.TiG_InitPacket.rRetract[4,3]:=	31.2	;	gImple.TiG_InitPacket.rExtend[4,3]:=	79.8	-20;	//E06Q1
gImple.TiG_InitPacket.rRetract[4,4]:=	31.5	;	gImple.TiG_InitPacket.rExtend[4,4]:=	80.2	-20;	//E06Q2
gImple.TiG_InitPacket.rRetract[4,5]:=	31.2	;	gImple.TiG_InitPacket.rExtend[4,5]:=	79.9	-20;	//E07Q1
gImple.TiG_InitPacket.rRetract[4,6]:=	30.5	;	gImple.TiG_InitPacket.rExtend[4,6]:=	79.1	-20;	//E07Q2
gImple.TiG_InitPacket.rRetract[4,7]:=	31.4	;	gImple.TiG_InitPacket.rExtend[4,7]:=	79.9	-20;	//E08Q1
gImple.TiG_InitPacket.rRetract[4,8]:=	32.3	;	gImple.TiG_InitPacket.rExtend[4,8]:=	80.8	-20;	//E08Q2
gImple.TiG_InitPacket.rRetract[5,1]:=	35.6	;	gImple.TiG_InitPacket.rExtend[5,1]:=	84.4	-20;	//E09Q1
gImple.TiG_InitPacket.rRetract[5,2]:=	33.0	;	gImple.TiG_InitPacket.rExtend[5,2]:=	82.1	-20;	//E09Q2
gImple.TiG_InitPacket.rRetract[5,3]:=	32.7	;	gImple.TiG_InitPacket.rExtend[5,3]:=	81.6	-20;	//E10Q1
gImple.TiG_InitPacket.rRetract[5,4]:=	33.9	;	gImple.TiG_InitPacket.rExtend[5,4]:=	82.4	-20;	//E10Q2
gImple.TiG_InitPacket.rRetract[5,5]:=	33.9	;	gImple.TiG_InitPacket.rExtend[5,5]:=	82.5	-20;	//E11Q1
gImple.TiG_InitPacket.rRetract[5,6]:=	33.7	;	gImple.TiG_InitPacket.rExtend[5,6]:=	82.9	-20;	//E11Q2
gImple.TiG_InitPacket.rRetract[5,7]:=	33.7	;	gImple.TiG_InitPacket.rExtend[5,7]:=	82.2	-20;	//E12Q1
gImple.TiG_InitPacket.rRetract[5,8]:=	33.7	;	gImple.TiG_InitPacket.rExtend[5,8]:=	82.2	-20;	//E12Q2
						
gImple.TiG_InitPacket.rRetract[6,1]:=	34.6	;	gImple.TiG_InitPacket.rExtend[6,1]:=	83.2	-20;	//E13Q
gImple.TiG_InitPacket.rRetract[6,2]:=	33.6	;	gImple.TiG_InitPacket.rExtend[6,2]:=	82.3	-20;	//E14Q
gImple.TiG_InitPacket.rRetract[6,3]:=	33.6	;	gImple.TiG_InitPacket.rExtend[6,3]:=	82.3	-20;	//E15Q
gImple.TiG_InitPacket.rRetract[6,4]:=	34.0	;	gImple.TiG_InitPacket.rExtend[6,4]:=	98.0	-30;	//E14L
	//gImple.TiG_InitPacket.rRetract[6,5]:=	32.8	;	gImple.TiG_InitPacket.rExtend[6,5]:=	96.2	-30;	//E15L
gImple.TiG_InitPacket.rRetract[6,5]:=	47.5	;	gImple.TiG_InitPacket.rExtend[6,5]:=	105.7	-30;	//E15L

gImple.TiG_InitPacket.rRetract[6,6]:=	35.2	;	gImple.TiG_InitPacket.rExtend[6,6]:=	98.8	-30;	//E13L
gImple.TiG_InitPacket.rRetract[6,7]:=	24.4	;	gImple.TiG_InitPacket.rExtend[6,7]:=	73.0	-25;	//E16L1
gImple.TiG_InitPacket.rRetract[6,8]:=	24.0	;	gImple.TiG_InitPacket.rExtend[6,8]:=	72.5	-25;	//E16L2
						
gImple.TiG_InitPacket.rRetract[7,1]:=	34.7	;	gImple.TiG_InitPacket.rExtend[7,1]:=	98.8	-30;	//E18L
gImple.TiG_InitPacket.rRetract[7,2]:=	37.1	;	gImple.TiG_InitPacket.rExtend[7,2]:=	100.8	-30;	//E19L
gImple.TiG_InitPacket.rRetract[7,3]:=	36.7	;	gImple.TiG_InitPacket.rExtend[7,3]:=	100.4	-30;	//E20L
gImple.TiG_InitPacket.rRetract[7,4]:=	34.1	;	gImple.TiG_InitPacket.rExtend[7,4]:=	98.1	-30;	//E21L
gImple.TiG_InitPacket.rRetract[7,5]:=	34.5	;	gImple.TiG_InitPacket.rExtend[7,5]:=	98.3	-30;	//E22L
gImple.TiG_InitPacket.rRetract[7,6]:=	35.3	;	gImple.TiG_InitPacket.rExtend[7,6]:=	98.9	-30;	//E23L
gImple.TiG_InitPacket.rRetract[7,7]:=	35.4	;	gImple.TiG_InitPacket.rExtend[7,7]:=	99.0	-30;	//E24L
gImple.TiG_InitPacket.rRetract[7,8]:=	35.2	;	gImple.TiG_InitPacket.rExtend[7,8]:=	98.9	-30;	//E25L
gImple.TiG_InitPacket.rRetract[7,9]:=	35.7	;	gImple.TiG_InitPacket.rExtend[7,9]:=	99.3	-30;	//E26L
gImple.TiG_InitPacket.rRetract[7,10]:=	35.0	;	gImple.TiG_InitPacket.rExtend[7,10]:=	83.6	-20;	//E17Q
gImple.TiG_InitPacket.rRetract[7,11]:=	33.9	;	gImple.TiG_InitPacket.rExtend[7,11]:=	82.5	-20;	//E18Q
gImple.TiG_InitPacket.rRetract[7,12]:=	32.9	;	gImple.TiG_InitPacket.rExtend[7,12]:=	81.3	-20;	//E19Q
gImple.TiG_InitPacket.rRetract[7,13]:=	33.5	;	gImple.TiG_InitPacket.rExtend[7,13]:=	82.0	-20;	//E20Q
gImple.TiG_InitPacket.rRetract[7,14]:=	34.9	;	gImple.TiG_InitPacket.rExtend[7,14]:=	83.3	-20;	//E21Q
gImple.TiG_InitPacket.rRetract[7,15]:=	34.9	;	gImple.TiG_InitPacket.rExtend[7,15]:=	83.7	-20;	//E22Q
gImple.TiG_InitPacket.rRetract[7,16]:=	33.5	;	gImple.TiG_InitPacket.rExtend[7,16]:=	82.0	-20;	//E23Q
gImple.TiG_InitPacket.rRetract[7,17]:=	34.0	;	gImple.TiG_InitPacket.rExtend[7,17]:=	82.5	-20;	//E24Q
gImple.TiG_InitPacket.rRetract[7,18]:=	34.6	;	gImple.TiG_InitPacket.rExtend[7,18]:=	83.2	-20;	//E25Q
gImple.TiG_InitPacket.rRetract[7,19]:=	36.1	;	gImple.TiG_InitPacket.rExtend[7,19]:=	84.6	-20;	//E26Q
gImple.TiG_InitPacket.rRetract[7,20]:=	24.5	;	gImple.TiG_InitPacket.rExtend[7,20]:=	73.0	-25;	//E17L1
gImple.TiG_InitPacket.rRetract[7,21]:=	23.7	;	gImple.TiG_InitPacket.rExtend[7,21]:=	72.3	-25;	//E17L2
gImple.TiG_InitPacket.rRetract[7,22]:=	23.7	;	gImple.TiG_InitPacket.rExtend[7,22]:=	72.4	-25;	//E27L1
gImple.TiG_InitPacket.rRetract[7,23]:=	24.5	;	gImple.TiG_InitPacket.rExtend[7,23]:=	73.2	-25;	//E27L2


(*------------------缩回位移标定值------------------------
gImple.TiG_InitPacket.rRetract[1,1]:=	23.8	;//E28L1
gImple.TiG_InitPacket.rRetract[1,2]:=	23.7	;//E28L2
gImple.TiG_InitPacket.rRetract[1,3]:=	33.3	;//E29L
gImple.TiG_InitPacket.rRetract[1,4]:=	34.3	;//E30L
gImple.TiG_InitPacket.rRetract[1,5]:=	32.6	;//E00L
gImple.TiG_InitPacket.rRetract[1,6]:=	33.0	;//E29Q
gImple.TiG_InitPacket.rRetract[1,7]:=	35.2	;//E30Q
gImple.TiG_InitPacket.rRetract[1,8]:=	32.5	;//E28Q
gImple.TiG_InitPacket.rRetract[1,9]:=	34.9	;//E01L
		
gImple.TiG_InitPacket.rRetract[2,1]:=	34.4	;//E02L
gImple.TiG_InitPacket.rRetract[2,2]:=	35.2	;//E03L
gImple.TiG_InitPacket.rRetract[2,3]:=	35.1	;//E04L
gImple.TiG_InitPacket.rRetract[2,4]:=	32.1	;//E05L
gImple.TiG_InitPacket.rRetract[2,5]:=	32.3	;//E06L
gImple.TiG_InitPacket.rRetract[2,6]:=	33.5	;//E07L
gImple.TiG_InitPacket.rRetract[2,7]:=	32.7	;//E08L
gImple.TiG_InitPacket.rRetract[2,8]:=	32.4	;//E09L
gImple.TiG_InitPacket.rRetract[2,9]:=	33.6	;//E10L
gImple.TiG_InitPacket.rRetract[2,10]:=	33.7	;//E11L
gImple.TiG_InitPacket.rRetract[2,11]:=	34.8	;//E12L
		
gImple.TiG_InitPacket.rRetract[3,1]:=	37.3	;//E01Q1
gImple.TiG_InitPacket.rRetract[3,2]:=	35.2	;//E01Q2
gImple.TiG_InitPacket.rRetract[3,3]:=	35.3	;//E02Q1
gImple.TiG_InitPacket.rRetract[3,4]:=	34.7	;//E02Q2
gImple.TiG_InitPacket.rRetract[3,5]:=	34.6	;//E03Q1
gImple.TiG_InitPacket.rRetract[3,6]:=	35.9	;//E03Q2
gImple.TiG_InitPacket.rRetract[3,7]:=	35.4	;//E04Q1
gImple.TiG_InitPacket.rRetract[3,8]:=	35.9	;//E04Q2
gImple.TiG_InitPacket.rRetract[4,1]:=	32.5	;//E05Q1
gImple.TiG_InitPacket.rRetract[4,2]:=	31.8	;//E05Q2
gImple.TiG_InitPacket.rRetract[4,3]:=	31.2	;//E06Q1
gImple.TiG_InitPacket.rRetract[4,4]:=	31.5	;//E06Q2
gImple.TiG_InitPacket.rRetract[4,5]:=	31.2	;//E07Q1
gImple.TiG_InitPacket.rRetract[4,6]:=	30.5	;//E07Q2
gImple.TiG_InitPacket.rRetract[4,7]:=	31.4	;//E08Q1
gImple.TiG_InitPacket.rRetract[4,8]:=	32.3	;//E08Q2
gImple.TiG_InitPacket.rRetract[5,1]:=	35.6	;//E09Q1
gImple.TiG_InitPacket.rRetract[5,2]:=	33.0	;//E09Q2
gImple.TiG_InitPacket.rRetract[5,3]:=	32.7	;//E10Q1
gImple.TiG_InitPacket.rRetract[5,4]:=	33.9	;//E10Q2
gImple.TiG_InitPacket.rRetract[5,5]:=	33.9	;//E11Q1
gImple.TiG_InitPacket.rRetract[5,6]:=	33.7	;//E11Q2
gImple.TiG_InitPacket.rRetract[5,7]:=	33.7	;//E12Q1
gImple.TiG_InitPacket.rRetract[5,8]:=	33.7	;//E12Q2
		
gImple.TiG_InitPacket.rRetract[6,1]:=	34.6	;//E13Q
gImple.TiG_InitPacket.rRetract[6,2]:=	33.6	;//E14Q
gImple.TiG_InitPacket.rRetract[6,3]:=	33.6	;//E15Q
gImple.TiG_InitPacket.rRetract[6,4]:=	34.0	;//E14L
gImple.TiG_InitPacket.rRetract[6,5]:=	32.8	;//E15L
gImple.TiG_InitPacket.rRetract[6,6]:=	35.2	;//E13L
gImple.TiG_InitPacket.rRetract[6,7]:=	24.4	;//E16L1
gImple.TiG_InitPacket.rRetract[6,8]:=	24.0	;//E16L2
		
gImple.TiG_InitPacket.rRetract[7,1]:=	34.7	;//E18L
gImple.TiG_InitPacket.rRetract[7,2]:=	37.1	;//E19L
gImple.TiG_InitPacket.rRetract[7,3]:=	36.7	;//E20L
gImple.TiG_InitPacket.rRetract[7,4]:=	34.1	;//E21L
gImple.TiG_InitPacket.rRetract[7,5]:=	34.5	;//E22L
gImple.TiG_InitPacket.rRetract[7,6]:=	35.3	;//E23L
gImple.TiG_InitPacket.rRetract[7,7]:=	35.4	;//E24L
gImple.TiG_InitPacket.rRetract[7,8]:=	35.2	;//E25L
gImple.TiG_InitPacket.rRetract[7,9]:=	35.7	;//E26L
gImple.TiG_InitPacket.rRetract[7,10]:=	35.0	;//E17Q
gImple.TiG_InitPacket.rRetract[7,11]:=	33.9	;//E18Q
gImple.TiG_InitPacket.rRetract[7,12]:=	32.9	;//E19Q
gImple.TiG_InitPacket.rRetract[7,13]:=	33.5	;//E20Q
gImple.TiG_InitPacket.rRetract[7,14]:=	34.9	;//E21Q
gImple.TiG_InitPacket.rRetract[7,15]:=	34.9	;//E22Q
gImple.TiG_InitPacket.rRetract[7,16]:=	33.5	;//E23Q
gImple.TiG_InitPacket.rRetract[7,17]:=	34.0	;//E24Q
gImple.TiG_InitPacket.rRetract[7,18]:=	34.6	;//E25Q
gImple.TiG_InitPacket.rRetract[7,19]:=	36.1	;//E26Q
gImple.TiG_InitPacket.rRetract[7,20]:=	24.5	;//E17L1
gImple.TiG_InitPacket.rRetract[7,21]:=	23.7	;//E17L2
gImple.TiG_InitPacket.rRetract[7,22]:=	23.7	;//E27L1
gImple.TiG_InitPacket.rRetract[7,23]:=	24.5	;//E27L2

//------------------伸出位移标定值------------------------
gImple.TiG_InitPacket.rExtend[1,1]:=	72.6	-25;	//E28L1
gImple.TiG_InitPacket.rExtend[1,2]:=	72.3	-25;	//E28L2
gImple.TiG_InitPacket.rExtend[1,3]:=	97.0	-30;	//E29L
gImple.TiG_InitPacket.rExtend[1,4]:=	98.1	-30;	//E30L
gImple.TiG_InitPacket.rExtend[1,5]:=	210.1	-30;//218.1;	//E00L
gImple.TiG_InitPacket.rExtend[1,6]:=	81.7	-20;	//E29Q
gImple.TiG_InitPacket.rExtend[1,7]:=	83.7	-20;	//E30Q
gImple.TiG_InitPacket.rExtend[1,8]:=	81.1	-20;	//E28Q
gImple.TiG_InitPacket.rExtend[1,9]:=	98.5	-30;	//E01L
			
gImple.TiG_InitPacket.rExtend[2,1]:=	98.0	-30;	//E02L
gImple.TiG_InitPacket.rExtend[2,2]:=	99.0	-30;	//E03L
gImple.TiG_InitPacket.rExtend[2,3]:=	98.7	-30;	//E04L
gImple.TiG_InitPacket.rExtend[2,4]:=	95.8	-30;	//E05L
gImple.TiG_InitPacket.rExtend[2,5]:=	95.9	-30;	//E06L
gImple.TiG_InitPacket.rExtend[2,6]:=	97.1	-30;	//E07L
gImple.TiG_InitPacket.rExtend[2,7]:=	96.3	-30;	//E08L
gImple.TiG_InitPacket.rExtend[2,8]:=	96.4	-30;	//E09L
gImple.TiG_InitPacket.rExtend[2,9]:=	96.3	-30;	//E10L
gImple.TiG_InitPacket.rExtend[2,10]:=	97.0	-30;	//E11L
gImple.TiG_InitPacket.rExtend[2,11]:=	97.0	-30;	//E12L
			
gImple.TiG_InitPacket.rExtend[3,1]:=	85.9	-20;	//E01Q1
gImple.TiG_InitPacket.rExtend[3,2]:=	83.6	-20;	//E01Q2
gImple.TiG_InitPacket.rExtend[3,3]:=	83.9	-20;	//E02Q1
gImple.TiG_InitPacket.rExtend[3,4]:=	83.3	-20;	//E02Q2
gImple.TiG_InitPacket.rExtend[3,5]:=	83.6	-20;	//E03Q1
gImple.TiG_InitPacket.rExtend[3,6]:=	84.3	-20;	//E03Q2
gImple.TiG_InitPacket.rExtend[3,7]:=	84.0	-20;	//E04Q1
gImple.TiG_InitPacket.rExtend[3,8]:=	84.4	-20;	//E04Q2
gImple.TiG_InitPacket.rExtend[4,1]:=	81.1	-20;	//E05Q1
gImple.TiG_InitPacket.rExtend[4,2]:=	80.3	-20;	//E05Q2
gImple.TiG_InitPacket.rExtend[4,3]:=	79.8	-20;	//E06Q1
gImple.TiG_InitPacket.rExtend[4,4]:=	80.2	-20;	//E06Q2
gImple.TiG_InitPacket.rExtend[4,5]:=	79.9	-20;	//E07Q1
gImple.TiG_InitPacket.rExtend[4,6]:=	79.1	-20;	//E07Q2
gImple.TiG_InitPacket.rExtend[4,7]:=	79.9	-20;	//E08Q1
gImple.TiG_InitPacket.rExtend[4,8]:=	80.8	-20;	//E08Q2
gImple.TiG_InitPacket.rExtend[5,1]:=	84.4	-20;	//E09Q1
gImple.TiG_InitPacket.rExtend[5,2]:=	82.1	-20;	//E09Q2
gImple.TiG_InitPacket.rExtend[5,3]:=	81.6	-20;	//E10Q1
gImple.TiG_InitPacket.rExtend[5,4]:=	82.4	-20;	//E10Q2
gImple.TiG_InitPacket.rExtend[5,5]:=	82.5	-20;	//E11Q1
gImple.TiG_InitPacket.rExtend[5,6]:=	82.9	-20;	//E11Q2
gImple.TiG_InitPacket.rExtend[5,7]:=	82.2	-20;	//E12Q1
gImple.TiG_InitPacket.rExtend[5,8]:=	82.2	-20;	//E12Q2
			
gImple.TiG_InitPacket.rExtend[6,1]:=	83.2	-20;	//E13Q
gImple.TiG_InitPacket.rExtend[6,2]:=	82.3	-20;	//E14Q
gImple.TiG_InitPacket.rExtend[6,3]:=	82.3	-20;	//E15Q
gImple.TiG_InitPacket.rExtend[6,4]:=	98.0	-30;	//E14L
gImple.TiG_InitPacket.rExtend[6,5]:=	96.2	-30;	//E15L
gImple.TiG_InitPacket.rExtend[6,6]:=	98.8	-30;	//E13L
gImple.TiG_InitPacket.rExtend[6,7]:=	73.0	-25;	//E16L1
gImple.TiG_InitPacket.rExtend[6,8]:=	72.5	-25;	//E16L2
			
gImple.TiG_InitPacket.rExtend[7,1]:=	98.8	-30;	//E18L
gImple.TiG_InitPacket.rExtend[7,2]:=	100.8	-30;	//E19L
gImple.TiG_InitPacket.rExtend[7,3]:=	100.4	-30;	//E20L
gImple.TiG_InitPacket.rExtend[7,4]:=	98.1	-30;	//E21L
gImple.TiG_InitPacket.rExtend[7,5]:=	98.3	-30;	//E22L
gImple.TiG_InitPacket.rExtend[7,6]:=	98.9	-30;	//E23L
gImple.TiG_InitPacket.rExtend[7,7]:=	99.0	-30;	//E24L
gImple.TiG_InitPacket.rExtend[7,8]:=	98.9	-30;	//E25L
gImple.TiG_InitPacket.rExtend[7,9]:=	99.3	-30;	//E26L
gImple.TiG_InitPacket.rExtend[7,10]:=	83.6	-20;	//E17Q
gImple.TiG_InitPacket.rExtend[7,11]:=	82.5	-20;	//E18Q
gImple.TiG_InitPacket.rExtend[7,12]:=	81.3	-20;	//E19Q
gImple.TiG_InitPacket.rExtend[7,13]:=	82.0	-20;	//E20Q
gImple.TiG_InitPacket.rExtend[7,14]:=	83.3	-20;	//E21Q
gImple.TiG_InitPacket.rExtend[7,15]:=	83.7	-20;	//E22Q
gImple.TiG_InitPacket.rExtend[7,16]:=	82.0	-20;	//E23Q
gImple.TiG_InitPacket.rExtend[7,17]:=	82.5	-20;	//E24Q
gImple.TiG_InitPacket.rExtend[7,18]:=	83.2	-20;	//E25Q
gImple.TiG_InitPacket.rExtend[7,19]:=	84.6	-20;	//E26Q
gImple.TiG_InitPacket.rExtend[7,20]:=	73.0	-25;	//E17L1
gImple.TiG_InitPacket.rExtend[7,21]:=	72.3	-25;	//E17L2
gImple.TiG_InitPacket.rExtend[7,22]:=	72.4	-25;	//E27L1
gImple.TiG_InitPacket.rExtend[7,23]:=	73.2	-25;	//E27L2
*)

FOR iVT:=1 TO 7 DO				//每个比例阀
	FOR iVT1:=1 TO aOil[iVT] DO	//比例阀中每个开关阀
		//-----------------------------------------------
		//gImple.TiG_InitPacket.rRetract[iVT,iVT1]:= 1;//校准数据需重新写入,按照上方注释
		//gImple.TiG_InitPacket.rExtend[iVT,iVT1]:= 200;
		//-----------------------------------------------
		gImple.PV_GroupTi.arrPV[iVT].sNum[iVT1].posVal.Retract:=gImple.TiG_InitPacket.rRetract[iVT,iVT1];
		gImple.PV_GroupTi.arrPV[iVT].sNum[iVT1].posVal.Extend:=gImple.TiG_InitPacket.rExtend[iVT,iVT1];		
		
	END_FOR
END_FOR

(*
FOR iVT:=1 TO 7 DO
	FOR iVT1:=1 TO aOil[iVT] DO
	END_FOR
END_FOR
*)


gImple.TiG_InitPacket.numHead[1,1]:=1;
gImple.TiG_InitPacket.numHead[1,2]:=3;
gImple.TiG_InitPacket.numHead[1,3]:=5;
gImple.TiG_InitPacket.numHead[1,4]:=6;
gImple.TiG_InitPacket.numHead[1,5]:=8;
gImple.TiG_InitPacket.numHead[1,6]:=9;
gImple.TiG_InitPacket.numHead[1,7]:=0;


gImple.TiG_InitPacket.numHead[2,1]:=1;
gImple.TiG_InitPacket.numHead[2,2]:=4;
gImple.TiG_InitPacket.numHead[2,3]:=5;
gImple.TiG_InitPacket.numHead[2,4]:=8;
gImple.TiG_InitPacket.numHead[2,5]:=9;
gImple.TiG_InitPacket.numHead[2,6]:=0;
gImple.TiG_InitPacket.numHead[2,7]:=0;

gImple.TiG_InitPacket.numHead[3,1]:=1;
gImple.TiG_InitPacket.numHead[4,1]:=1;
gImple.TiG_InitPacket.numHead[5,1]:=1;

FOR iVT:=3 TO 5 DO
	FOR iVT1:=2 TO 7 DO
		gImple.TiG_InitPacket.numHead[iVT,iVT1]:=0;
	END_FOR
END_FOR

gImple.TiG_InitPacket.numHead[6,1]:=1;
gImple.TiG_InitPacket.numHead[6,2]:=3;
gImple.TiG_InitPacket.numHead[6,3]:=4;
gImple.TiG_InitPacket.numHead[6,4]:=6;
gImple.TiG_InitPacket.numHead[6,5]:=7;
gImple.TiG_InitPacket.numHead[6,6]:=0;
gImple.TiG_InitPacket.numHead[6,7]:=0;

gImple.TiG_InitPacket.numHead[7,1]:=1;
gImple.TiG_InitPacket.numHead[7,2]:=5;
gImple.TiG_InitPacket.numHead[7,3]:=6;
gImple.TiG_InitPacket.numHead[7,4]:=10;
gImple.TiG_InitPacket.numHead[7,5]:=15;
gImple.TiG_InitPacket.numHead[7,6]:=20;
gImple.TiG_InitPacket.numHead[7,7]:=22;

//----------

gImple.TiG_InitPacket.numTail[1,1]:=2;
gImple.TiG_InitPacket.numTail[1,2]:=4;
gImple.TiG_InitPacket.numTail[1,3]:=5;
gImple.TiG_InitPacket.numTail[1,4]:=7;
gImple.TiG_InitPacket.numTail[1,5]:=8;
gImple.TiG_InitPacket.numTail[1,6]:=9;
gImple.TiG_InitPacket.numTail[1,7]:=0;


gImple.TiG_InitPacket.numTail[2,1]:=3;
gImple.TiG_InitPacket.numTail[2,2]:=4;
gImple.TiG_InitPacket.numTail[2,3]:=7;
gImple.TiG_InitPacket.numTail[2,4]:=8;
gImple.TiG_InitPacket.numTail[2,5]:=11;
gImple.TiG_InitPacket.numTail[2,6]:=0;
gImple.TiG_InitPacket.numTail[2,7]:=0;

gImple.TiG_InitPacket.numTail[3,1]:=8;
gImple.TiG_InitPacket.numTail[4,1]:=8;
gImple.TiG_InitPacket.numTail[5,1]:=8;

FOR iVT:=3 TO 5 DO
	FOR iVT1:=2 TO 7 DO
		gImple.TiG_InitPacket.numTail[iVT,iVT1]:=0;
	END_FOR
END_FOR

gImple.TiG_InitPacket.numTail[6,1]:=2;
gImple.TiG_InitPacket.numTail[6,2]:=3;
gImple.TiG_InitPacket.numTail[6,3]:=5;
gImple.TiG_InitPacket.numTail[6,4]:=6;
gImple.TiG_InitPacket.numTail[6,5]:=8;
gImple.TiG_InitPacket.numTail[6,6]:=0;
gImple.TiG_InitPacket.numTail[6,7]:=0;

gImple.TiG_InitPacket.numTail[7,1]:=4;
gImple.TiG_InitPacket.numTail[7,2]:=5;
gImple.TiG_InitPacket.numTail[7,3]:=9;
gImple.TiG_InitPacket.numTail[7,4]:=14;
gImple.TiG_InitPacket.numTail[7,5]:=19;
gImple.TiG_InitPacket.numTail[7,6]:=21;
gImple.TiG_InitPacket.numTail[7,7]:=23;

FOR iVT:=1 TO 7 DO				//每个比例阀
	FOR iVT1:=1 TO aNo[iVT] DO	//比例阀中每个开关阀
		IF gImple.TiG_InitPacket.numHead[iVT,iVT1]>0 THEN
			
			gImple.TiG_InitPacket.numInColumn[iVT,iVT1]:= gImple.TiG_InitPacket.numTail[iVT,iVT1]-gImple.TiG_InitPacket.numHead[iVT,iVT1]+1;
			
		END_IF
	END_FOR	
END_FOR

gImple.PV_GroupTi.arrAddtion[1].sPlateStatus.sSensor.Extend:=	105;
gImple.PV_GroupTi.arrAddtion[1].sPlateStatus.sSensor.Retract:=	20;
gImple.PV_GroupTi.arrAddtion[2].sPlateStatus.sSensor.Extend:=	98.1;
gImple.PV_GroupTi.arrAddtion[2].sPlateStatus.sSensor.Retract:=	25.7;
END_ACTION

METHOD statusPercentCalcTi	:REAL
VAR_INPUT
	psTiG				:POINTER TO propValveModule_Ti;	//天轨结构体

	iDTENum				:INT;							//天轨比例阀组号
	iIndex				:INT;							//比例阀组内索引
END_VAR
VAR
	rTotal				:REAL;
	rGone				:REAL;
END_VAR

IF psTiG^.arrPV[iDTENum].sNum[iIndex].posVal.Current > 3.0 THEN
	rGone:=psTiG^.arrPV[iDTENum].sNum[iIndex].posVal.Current-psTiG^.arrPV[iDTENum].sNum[iIndex].posVal.Retract;
	rTotal:=psTiG^.arrPV[iDTENum].sNum[iIndex].posVal.Extend-psTiG^.arrPV[iDTENum].sNum[iIndex].posVal.Retract;
	
	statusPercentCalcTi:=rGone/rTotal*100;
END_IF
END_METHOD

METHOD cmdDeliverTi : BOOL
VAR_INPUT
	
END_VAR
VAR
	eCommand				:cmdStat;
	arrOBUSP				:ARRAY[1..8] OF OilBlockUnit_Status_PosVal;
	fbCheckGrop				:ARRAY[1..7,1..7] OF checkoilGropisDoneX8;
	iCount					:UINT;	
	iCntErr					:UINT:=250*6;			//超时时间1s=250
	iTemp					:INT;

END_VAR

FOR iVT:=1 TO 7 DO
	IF gUI.TiG.arrPV[iVT].bPVD_enable THEN
		gImple.PV_GroupTi.arrPV[iVT].percenVal:=REAL_TO_WORD(gUI.TiG.arrPV[iVT].rPVDPercent* 65535/100.0);
	ELSE
		gImple.PV_GroupTi.arrPV[iVT].percenVal:=0;
	END_IF
END_FOR

FOR iVT:=1 TO 7 DO				//每个比例阀
	
	FOR iVT1:=1 TO aNo[iVT] DO	//比例阀中每个开关阀
		//取出计数值
		iCount:=gImple.PV_GroupTi.arrPV[iVT].iCntErr[iVT1];
		//根据按钮判断指令
		IF gUI.TiG.arrPV[iVT].sColumn[iVT1].bExtend<>gUI.TiG.arrPV[iVT].sColumn[iVT1].bRetract THEN
			gImple.PV_GroupTi.arrPV[iVT].sColumn[iVT1].eStat:=cmdStat.eRun;
			IF gUI.TiG.arrPV[iVT].sColumn[iVT1].bExtend THEN
				eCommand:=cmdStat.cExtend;
				gUI.TiG.arrPV[iVT].sColumn[iVT1].cmdLast:=cmdStat.cExtend;
			END_IF
			IF gUI.TiG.arrPV[iVT].sColumn[iVT1].bRetract THEN
				eCommand:=cmdStat.cRetract;
				gUI.TiG.arrPV[iVT].sColumn[iVT1].cmdLast:=cmdStat.cRetract;
			END_IF
		ELSE
			eCommand:=cmdStat.cStop;
			IF gUI.TiG.arrPV[iVT].sColumn[iVT1].bExtend THEN
				iCount:=0;
				gImple.PV_GroupTi.arrPV[iVT].sColumn[iVT1].eStat:=cmdStat.eRun;
				CASE gUI.TiG.arrPV[iVT].sColumn[iVT1].cmdLast OF
					cmdStat.cExtend:
						gUI.TiG.arrPV[iVT].sColumn[iVT1].bStop:=FALSE;
						gUI.TiG.arrPV[iVT].sColumn[iVT1].bExtend:=FALSE;
						gUI.TiG.arrPV[iVT].sColumn[iVT1].bRetract:=TRUE;
						eCommand:=cmdStat.cRetract;
					cmdStat.cRetract:
						gUI.TiG.arrPV[iVT].sColumn[iVT1].bStop:=FALSE;
						gUI.TiG.arrPV[iVT].sColumn[iVT1].bExtend:=TRUE;
						gUI.TiG.arrPV[iVT].sColumn[iVT1].bRetract:=FALSE;
						eCommand:=cmdStat.cExtend;
				END_CASE
			END_IF
		END_IF

		IF gUI.TiG.arrPV[iVT].sColumn[iVT1].bStop THEN
			eCommand:=cmdStat.cStop;
		END_IF
		//根据指令判断每个开关阀下的油缸状态是否已经到位
		FOR iTemp:= 1 TO 8 DO
			arrOBUSP[iTemp]:=GetPositionValueOfUnit8(ADR(gImple.PV_GroupTi),ADR(gImple.TiG_InitPacket),iVT,iVT1,iTemp);
		END_FOR
		fbCheckGrop[iVT,iVT1](
			cmdAct		:=eCommand,
			arrPosVal	:=arrOBUSP,
			bFetch		 =>
		);
		
		IF fbCheckGrop[iVT,iVT1].bFetch=TRUE THEN
			//已经到位则清零计数器
			iCount:=0;
			IF gImple.PV_GroupTi.arrPV[iVT].sColumn[iVT1].eStat<>cmdStat.eError THEN
				//正常态油缸指令复位
				gUI.TiG.arrPV[iVT].sColumn[iVT1].bStop:=FALSE;
				gUI.TiG.arrPV[iVT].sColumn[iVT1].bExtend:=FALSE;
				gUI.TiG.arrPV[iVT].sColumn[iVT1].bRetract:=FALSE;	
				cmdExecuteT(ADR(gImple.PV_GroupTi),iVT,iVT1,cmdStat.cStop);
				//判断每个开关阀的总状态（伸出or收回）	 
				fbCheckGrop[iVT,iVT1](cmdAct:=cmdStat.cExtend,arrPosVal:=arrOBUSP);
				IF fbCheckGrop[iVT,iVT1].bFetch=TRUE THEN
					gImple.PV_GroupTi.arrPV[iVT].sColumn[iVT1].eStat:=cmdStat.Extend_Done;
				END_IF
				fbCheckGrop[iVT,iVT1](cmdAct:=cmdStat.cRetract,arrPosVal:=arrOBUSP);
				IF fbCheckGrop[iVT,iVT1].bFetch=TRUE THEN
					gImple.PV_GroupTi.arrPV[iVT].sColumn[iVT1].eStat:=cmdStat.Retract_Done;
				END_IF			
				//都不是则为Normal态
				IF gImple.PV_GroupTi.arrPV[iVT].sColumn[iVT1].eStat<>cmdStat.Retract_Done AND gImple.PV_GroupTi.arrPV[iVT].sColumn[iVT1].eStat<>cmdStat.Extend_Done THEN
					gImple.PV_GroupTi.arrPV[iVT].sColumn[iVT1].eStat:=cmdStat.eNormal;
				END_IF
				
			END_IF
		ELSE
			iCount:= iCount +1;
			gImple.PV_GroupTi.arrPV[iVT].sColumn[iVT1].eStat:=cmdStat.eRun;
			cmdExecuteT(ADR(gImple.PV_GroupTi),iVT,iVT1,eCommand);
		END_IF
		
		IF iCount>=iCntErr THEN
			//错误态油缸指令复位
			gImple.PV_GroupTi.arrPV[iVT].sColumn[iVT1].eStat:=cmdStat.eError;
			gUI.TiG.arrPV[iVT].sColumn[iVT1].bStop:=FALSE;
			gUI.TiG.arrPV[iVT].sColumn[iVT1].bExtend:=FALSE;
			gUI.TiG.arrPV[iVT].sColumn[iVT1].bRetract:=FALSE;
			cmdExecuteT(ADR(gImple.PV_GroupTi),iVT,iVT1,cmdStat.cStop);
		END_IF		
		gImple.PV_GroupTi.arrPV[iVT].iCntErr[iVT1]:=iCount;
		
	END_FOR
END_FOR
END_METHOD

METHOD cmdDeliverPlate : BOOL
VAR_INPUT
END_VAR
VAR
	eCommand				:cmdStat;
	arrOBUSP				:ARRAY[1..8] OF OilBlockUnit_Status_PosVal;
	fbCheckGrop				:ARRAY[1..2] OF checkoilGropisDoneX8;
	iCount					:UINT;	
	iCntErr					:UINT:=250*6;			//超时时间1s=250
	iTemp					:INT;

END_VAR

FOR iVT:=1 TO 2 DO				//2个挡板
		//取出计数值
		iCount:=gImple.PV_GroupTi.arrAddtion[iVT].sPlateStatus.iCnt;
		//根据按钮判断指令
		IF gUI.TiG.arrPlate[iVT].sCmd.bExtend<>gUI.TiG.arrPlate[iVT].sCmd.bRetract THEN
			gImple.PV_GroupTi.arrAddtion[iVT].sPlateStatus.eStat:=cmdStat.eRun;
			IF gUI.TiG.arrPlate[iVT].sCmd.bExtend THEN
				eCommand:=cmdStat.cExtend;
				gUI.TiG.arrPlate[iVT].sCmd.cmdLast:=cmdStat.cExtend;
			END_IF
			IF gUI.TiG.arrPlate[iVT].sCmd.bRetract THEN
				eCommand:=cmdStat.cRetract;	
				gUI.TiG.arrPlate[iVT].sCmd.cmdLast:=cmdStat.cRetract;
			END_IF
		ELSE
			eCommand:=cmdStat.cStop;
			IF gUI.TiG.arrPlate[iVT].sCmd.bExtend THEN
				iCount:=0;
				gImple.PV_GroupTi.arrAddtion[iVT].sPlateStatus.eStat:=cmdStat.eRun;
				CASE gUI.TiG.arrPlate[iVT].sCmd.cmdLast OF
					cmdStat.cExtend:
						gUI.TiG.arrPlate[iVT].sCmd.bStop:=FALSE;
						gUI.TiG.arrPlate[iVT].sCmd.bExtend:=FALSE;
						gUI.TiG.arrPlate[iVT].sCmd.bRetract:=TRUE;
						eCommand:=cmdStat.cRetract;
					cmdStat.cRetract:
						gUI.TiG.arrPlate[iVT].sCmd.bStop:=FALSE;
						gUI.TiG.arrPlate[iVT].sCmd.bExtend:=TRUE;
						gUI.TiG.arrPlate[iVT].sCmd.bRetract:=FALSE;
						eCommand:=cmdStat.cExtend;

				END_CASE
			END_IF
		END_IF
		
		IF gUI.TiG.arrPV[iVT].sColumn[iVT1].bStop THEN
			eCommand:=cmdStat.cStop;
		END_IF	
		
		//根据指令判断每个开关阀下的油缸状态是否已经到位
		arrOBUSP[1].Current:=gImple.PV_GroupTi.arrAddtion[iVT].sPlateStatus.sSensor.Current;
		arrOBUSP[1].Extend:=gImple.PV_GroupTi.arrAddtion[iVT].sPlateStatus.sSensor.Extend;
		arrOBUSP[1].Retract:=gImple.PV_GroupTi.arrAddtion[iVT].sPlateStatus.sSensor.Retract;
		arrOBUSP[2].Current:=0;	arrOBUSP[2].Extend:=0;arrOBUSP[2].Retract:=0;
		fbCheckGrop[iVT](
			cmdAct		:=eCommand,
			arrPosVal	:=arrOBUSP,
			bFetch		 =>
		);
		
		IF fbCheckGrop[iVT].bFetch=TRUE THEN
			//已经到位则清零计数器
			iCount:=0;
			IF gImple.PV_GroupTi.arrAddtion[iVT].sPlateStatus.eStat<>cmdStat.eError THEN
				//正常态油缸指令复位
				gUI.TiG.arrPlate[iVT].sCmd.bStop:=FALSE;
				gUI.TiG.arrPlate[iVT].sCmd.bExtend:=FALSE;
				gUI.TiG.arrPlate[iVT].sCmd.bRetract:=FALSE;	
				cmdExecutePlate(ADR(gImple.PV_GroupTi),iVT,cmdStat.cStop);
				//判断每个开关阀的总状态（伸出or收回）	 
				fbCheckGrop[iVT](cmdAct:=cmdStat.cExtend,arrPosVal:=arrOBUSP);
				IF fbCheckGrop[iVT].bFetch=TRUE THEN
					gImple.PV_GroupTi.arrAddtion[iVT].sPlateStatus.eStat:=cmdStat.Extend_Done;
				END_IF
				fbCheckGrop[iVT](cmdAct:=cmdStat.cRetract,arrPosVal:=arrOBUSP);
				IF fbCheckGrop[iVT].bFetch=TRUE THEN
					gImple.PV_GroupTi.arrAddtion[iVT].sPlateStatus.eStat:=cmdStat.Retract_Done;
				END_IF			
				//都不是则为Normal态
				IF gImple.PV_GroupTi.arrAddtion[iVT].sPlateStatus.eStat<>cmdStat.Retract_Done AND gImple.PV_GroupTi.arrAddtion[iVT].sPlateStatus.eStat<>cmdStat.Extend_Done THEN
					gImple.PV_GroupTi.arrAddtion[iVT].sPlateStatus.eStat:=cmdStat.eNormal;
				END_IF
				
			END_IF
		ELSE
			iCount:= iCount +1;
			gImple.PV_GroupTi.arrAddtion[iVT].sPlateStatus.eStat:=cmdStat.eRun;
			cmdExecutePlate(ADR(gImple.PV_GroupTi),iVT,eCommand);

		END_IF
		
		IF iCount>=iCntErr THEN
			//错误态油缸指令复位
			gImple.PV_GroupTi.arrPV[iVT].sColumn[iVT1].eStat:=cmdStat.eError;
			gUI.TiG.arrPV[iVT].sColumn[iVT1].bStop:=FALSE;
			gUI.TiG.arrPV[iVT].sColumn[iVT1].bExtend:=FALSE;
			gUI.TiG.arrPV[iVT].sColumn[iVT1].bRetract:=FALSE;
			cmdExecutePlate(ADR(gImple.PV_GroupTi),iVT,cmdStat.cStop);
		END_IF		
		gImple.PV_GroupTi.arrAddtion[iVT].sPlateStatus.iCnt:=iCount;
		

END_FOR
END_METHOD

METHOD cmdDeliverManual :BOOL
VAR_INPUT
END_VAR
VAR
	eCommand				:cmdStat;

END_VAR
FOR iVT:=1 TO 7 DO
	IF gUI.TiG.arrPV[iVT].bPVD_enable THEN
		gImple.PV_GroupTi.arrPV[iVT].percenVal:=REAL_TO_WORD(gUI.TiG.arrPV[iVT].rPVDPercent* 65535/100.0);
	ELSE
		gImple.PV_GroupTi.arrPV[iVT].percenVal:=0;
	END_IF
END_FOR

FOR iVT:=1 TO 7 DO				//每个比例阀
	FOR iVT1:=1 TO aNo[iVT] DO	//比例阀中每个开关阀
		//根据按钮判断指令
		IF gUI.TiG.arrPV[iVT].sColumn[iVT1].bExtend<>gUI.TiG.arrPV[iVT].sColumn[iVT1].bRetract THEN
			IF gUI.TiG.arrPV[iVT].sColumn[iVT1].bExtend THEN
				eCommand:=cmdStat.cExtend;
			END_IF
			IF gUI.TiG.arrPV[iVT].sColumn[iVT1].bRetract THEN
				eCommand:=cmdStat.cRetract;
			END_IF
		ELSE
			eCommand:=cmdStat.cStop;
		END_IF
		IF gUI.TiG.arrPV[iVT].sColumn[iVT1].bStop THEN
			eCommand:=cmdStat.cStop;
		END_IF
		cmdExecuteT(ADR(gImple.PV_GroupTi),iVT,iVT1,eCommand);
	END_FOR
END_FOR
	
FOR iVT:=1 TO 2 DO
	IF gUI.TiG.arrPlate[iVT].sCmd.bExtend<>gUI.TiG.arrPlate[iVT].sCmd.bRetract THEN
		IF gUI.TiG.arrPlate[iVT].sCmd.bExtend THEN
			eCommand:=cmdStat.cExtend;
		END_IF
		IF gUI.TiG.arrPlate[iVT].sCmd.bRetract THEN
			eCommand:=cmdStat.cRetract;	
		END_IF
	ELSE
		eCommand:=cmdStat.cStop;	
	END_IF
	IF gUI.TiG.arrPV[iVT].sColumn[iVT1].bStop THEN
		eCommand:=cmdStat.cStop;
	END_IF	
	cmdExecutePlate(ADR(gImple.PV_GroupTi),iVT,eCommand);
END_FOR
END_METHOD

END_PROGRAM

// Device/Application/public_datum/cmdcheck/fUICmdDetect
FUNCTION fUICmdDetect : BOOL
VAR_INPUT
	psUITi			:POINTER TO UICell_OilBlock_Ti;
END_VAR
VAR
	bCmdDetected	:BOOL;
	iV1				:INT;
	iV2				:INT;
END_VAR
VAR CONSTANT
	aNo		:ARRAY [1..7] OF INT :=[6, 5,1,1,1,5, 7];		//每个比例阀下开关阀的数量(天轨):arrMappingRealNumTiG
END_VAR

bCmdDetected:=FALSE;


FOR iV1:=1 TO 7 DO				//每个比例阀
	FOR iV2:=1 TO aNo[iV1] DO	//比例阀中每个开关阀
		IF psUITi^.arrPV[iV1].sColumn[iV2].bExtend OR psUITi^.arrPV[iV1].sColumn[iV2].bRetract THEN
			bCmdDetected:=TRUE;
		END_IF
	END_FOR	
END_FOR

IF psUITi^.arrPlate[1].sCmd.bExtend OR psUITi^.arrPlate[1].sCmd.bRetract THEN
	bCmdDetected:=TRUE;
END_IF
IF psUITi^.arrPlate[2].sCmd.bExtend OR psUITi^.arrPlate[2].sCmd.bRetract THEN
	bCmdDetected:=TRUE;
END_IF

fUICmdDetect:=bCmdDetected;

END_FUNCTION

// Device/Application/public_datum/cmdcheck/percentCalc
FUNCTION_BLOCK percentCalc
VAR_INPUT
	rInput				:REAL;
	rExtend				:REAL;
	rRetract			:REAL;
END_VAR
VAR_OUTPUT
	rOut				:REAL;
END_VAR
VAR
	rTotal				:REAL;
	rGone				:REAL;
END_VAR

IF rInput>1 THEN
	rGone:=rInput-rRetract;
	rTotal:=rExtend-rRetract;
	rOut:=rGone/rTotal*100;
END_IF

END_FUNCTION_BLOCK

// Device/Application/public_datum/cmdcheck/GetPositionValueOfUnit8
FUNCTION GetPositionValueOfUnit8 : OilBlockUnit_Status_PosVal
VAR_INPUT
	psPVTi			: POINTER TO propValveModule_Ti;
	psTipakt		: POINTER TO OilBlockUnit_RangeRec;
	iVT				: INT;	//比例阀序号
	iVT1			: INT;	//比例阀下的开关阀序号
	iSequence		: INT;	//充入八个结构体数组中的索引值(1~8)

END_VAR
VAR

	iSum			:INT;	//每个开关阀下的油缸数量
	iIndexHead		:INT;	//要查找的油缸索引头号位置
	iIndexFind		:INT;	//要查找的油缸索引值
	//iIndexTail		:INT;	//要查找的油缸索引尾号位置
	//iTemp			:INT;
	
END_VAR

//获取油缸个数
iSum:= psTipakt^.numInColumn[iVT,iVT1];

IF iSum < iSequence THEN
	GetPositionValueOfUnit8.Extend	:= 0;
	GetPositionValueOfUnit8.Retract	:= 0;
	GetPositionValueOfUnit8.Current := 0;
ELSE
	iIndexFind :=  psTipakt^.numHead[iVT,iVT1] + iSequence -1;
	GetPositionValueOfUnit8.Extend	:= psPVTi^.arrPV[iVT].sNum[iIndexFind].posVal.Extend;
	GetPositionValueOfUnit8.Retract	:= psPVTi^.arrPV[iVT].sNum[iIndexFind].posVal.Retract;
	GetPositionValueOfUnit8.Current	:= psPVTi^.arrPV[iVT].sNum[iIndexFind].posVal.Current;


END_IF














(*
//获取油缸状态
FOR iTemp := 1 TO iOilNum DO
	GetArrayOfPositionValue[iTemp].Extend  :=psPVTi^.arrPV[iVT].sNum[iIndexHead+iTemp-1].posVal.Extend;
	GetArrayOfPositionValue[iTemp].Current :=psPVTi^.arrPV[iVT].sNum[iIndexHead+iTemp-1].posVal.Current;
	GetArrayOfPositionValue[iTemp].Retract :=psPVTi^.arrPV[iVT].sNum[iIndexHead+iTemp-1].posVal.Retract;
END_FOR
//将剩余变量置0
IF iOilNum<8 THEN
	FOR iTemp := (iOilNum+1) TO 8 DO
		GetArrayOfPositionValue[iTemp].Extend  :=0;
		GetArrayOfPositionValue[iTemp].Current :=0;
		GetArrayOfPositionValue[iTemp].Retract :=0;
	END_FOR
END_IF
*)

END_FUNCTION

// Device/Application/rail_ceiling/cmdExecuteT
FUNCTION cmdExecuteT : BOOL
VAR_INPUT
	psPVTi			: POINTER TO propValveModule_Ti;
	iVT				:INT;
	iVTN			:INT;
	iCmd			:cmdStat;		
END_VAR
VAR
	
END_VAR


CASE iCmd OF
	cmdStat.cStop:
		psPVTi^.arrPV[iVT].sColumn[iVTN].bE_Open:=0;
		psPVTi^.arrPV[iVT].sColumn[iVTN].bR_Open:=0;
	cmdStat.cRetract:
		psPVTi^.arrPV[iVT].sColumn[iVTN].bE_Open:=0;
		psPVTi^.arrPV[iVT].sColumn[iVTN].bR_Open:=1;
	cmdStat.cExtend:
		psPVTi^.arrPV[iVT].sColumn[iVTN].bE_Open:=1;
		psPVTi^.arrPV[iVT].sColumn[iVTN].bR_Open:=0;
END_CASE

END_FUNCTION

// Device/Application/public_datum/cmdcheck/checkoilGropisDoneX8
FUNCTION_BLOCK checkoilGropisDoneX8
VAR_INPUT
	cmdAct		:cmdStat;
	arrPosVal	:ARRAY  [1..8] OF OilBlockUnit_Status_PosVal;
END_VAR
VAR_OUTPUT
	bFetch		:BOOL;
END_VAR
VAR
	outStat			:ARRAY[1..8] OF OilBlockUnit_Status_Loc;
	//arrCheckUnit	:ARRAY[1..8] OF  checkoilUnit;
	iCheck			:INT;
	iNum			:INT;				//有值的位移传感器值
	iTemp			:INT;
	bAllDone		:BOOL;
END_VAR

//判断有多少个油缸需状态检测，Extend==0||Retract==0||Current==0的不检测
iNum:=0;
FOR iTemp :=1 TO 8 DO
	IF arrPosVal[iTemp].Extend <> 0 THEN
		iNum:=iNum+1;
	END_IF
END_FOR


//对要动作的油缸进行位置检测
(*
FOR iCheck:=1 TO iNum DO
	arrCheckUnit[iCheck]
	(
		rExtend	:=arrPosVal[iCheck].Extend,
		rRetract:=arrPosVal[iCheck].Retract,
		rCurrent:=arrPosVal[iCheck].Current,
		rError	:=2.0,
		outStat	 =>
	);
END_FOR
*)
FOR iCheck:=1 TO iNum DO
	outStat[iCheck]	:=fGetUnitStat(arrPosVal[iCheck].Extend,arrPosVal[iCheck].Retract,arrPosVal[iCheck].Current,2.0);
END_FOR

bAllDone:=TRUE;

	//有一个未到指令位置则未完成
	CASE cmdAct OF 
		cmdStat.cExtend:
			FOR iCheck:=1 TO iNum DO
				IF outStat[iCheck]<>OilBlockUnit_Status_Loc.eExtended THEN
					bAllDone:=FALSE;
				END_IF
			END_FOR
		cmdStat.cRetract:
			FOR iCheck:=1 TO iNum DO
				IF outStat[iCheck]<>OilBlockUnit_Status_Loc.eRetracted THEN
					bAllDone:=FALSE;
				END_IF
			END_FOR	
		cmdStat.cStop:
			
	END_CASE

IF bAllDone THEN
	bFetch	:= TRUE;
ELSE
	bFetch	:= FALSE;
END_IF

END_FUNCTION_BLOCK

// Device/Application/public_datum/cmdcheck/fGetUnitStat
FUNCTION fGetUnitStat : OilBlockUnit_Status_Loc
VAR_INPUT
	rExtend 		:REAL;    //伸出位置
	rRetract   		:REAL;    //收回位置
	rCurrent 		:REAL;    //当前位置
	rError			:REAL;	  //误差范围
END_VAR
VAR
	tempStat		:OilBlockUnit_Status_Loc;		//输出状态
END_VAR

IF rCurrent > 1 THEN						 //实际位置总是大于1mm的

	IF (rCurrent<rRetract+rError) THEN
		tempStat:=OilBlockUnit_Status_Loc.eRetracted;
	ELSIF (rCurrent>rExtend-rError) THEN
		tempStat:=OilBlockUnit_Status_Loc.eExtended;
	ELSE
		tempStat:=OilBlockUnit_Status_Loc.eRunning;
	END_IF
	
(*	
	IF  ABS( rCurrent - rRetract)< rError THEN	//rCurrent<rRetract+rError
		tempStat:=OilBlockUnit_Status_Loc.eRetracted;
	ELSIF ABS( rCurrent - rExtend)< rError THEN	//rCurrent>rExtend-rError
		tempStat:=OilBlockUnit_Status_Loc.eExtended;
	ELSE
		tempStat:=OilBlockUnit_Status_Loc.eRunning;
	END_IF
*)	
END_IF

	

fGetUnitStat:=tempStat;

END_FUNCTION

// Device/Application/public_datum/cmdcheck/checkoilUnit
FUNCTION_BLOCK checkoilUnit
VAR_INPUT
	rExtend 		:REAL;    //伸出位置
	rRetract   		:REAL;    //收回位置
	rCurrent 		:REAL;    //当前位置
	rError			:REAL;	  //误差范围
END_VAR
VAR_OUTPUT
	outStat			:OilBlockUnit_Status_Loc;		//输出状态
END_VAR
VAR
	iCntE			:UINT:=0;			//伸出检测计数
	iCntR			:UINT:=0;			//收回检测计数
	tempStat		:OilBlockUnit_Status_Loc;		//输出状态
END_VAR

//?ms调用1次
(*
IF rCurrent > 1 THEN						 //实际位置总是大于1mm的
	IF (rRetract+rError<=rCurrent) THEN
		iCntE:=0;
		iCntR:=iCntR+1;
	ELSIF (rCurrent<=rExtend-rError) THEN
		iCntE:=iCntE+1;
		iCntR:=0;
	ELSE
		iCntE:=0;
		iCntR:=0;
	END_IF
	
	IF iCntE>=10 THEN
		iCntE:=10;
		tempStat:=OilBlockUnit_Status_Loc.eExtended;
	ELSIF iCntR>=10 THEN
		iCntR:=10;
		tempStat:=OilBlockUnit_Status_Loc.eRetracted;
	ELSE
		tempStat:=OilBlockUnit_Status_Loc.eRunning;
	END_IF
ELSE
	iCntE:=0;
	iCntR:=0;
	tempStat:=OilBlockUnit_Status_Loc.eUnknow;
END_IF
*)
IF rCurrent > 1 THEN						 //实际位置总是大于1mm的
	IF (rRetract+rError<=rCurrent) THEN
		tempStat:=OilBlockUnit_Status_Loc.eRetracted;
	ELSIF (rCurrent<=rExtend-rError) THEN
		tempStat:=OilBlockUnit_Status_Loc.eExtended;
	ELSE
		tempStat:=OilBlockUnit_Status_Loc.eRunning;
	END_IF

END_IF

	

outStat:=tempStat;

END_FUNCTION_BLOCK

// Device/Application/rail_plate/cmdExecutePlate
FUNCTION cmdExecutePlate : BOOL

VAR_INPUT
	psPVTi			: POINTER TO propValveModule_Ti;
	iVT				:INT;
	iCmd			:cmdStat;		
END_VAR

VAR
END_VAR

CASE iCmd OF
	cmdStat.cStop:
		psPVTi^.arrAddtion[iVT].sPlateCtrl.bExtend:=0;
		psPVTi^.arrAddtion[iVT].sPlateCtrl.bRetract:=0;
	cmdStat.cRetract:
		psPVTi^.arrAddtion[iVT].sPlateCtrl.bExtend:=0;
		psPVTi^.arrAddtion[iVT].sPlateCtrl.bRetract:=1;
	cmdStat.cExtend:
		psPVTi^.arrAddtion[iVT].sPlateCtrl.bExtend:=1;
		psPVTi^.arrAddtion[iVT].sPlateCtrl.bRetract:=0;

END_CASE

END_FUNCTION

// Device/Application/dataUpload/tcpUploader
PROGRAM tcpUploader
VAR
	destIp 			:STRING:='172.168.31.57';
	destPort 		:UINT:= 61558;
	tcpConnector	:tcpUpload;
	
	myData 			:ARRAY[1..1024]OF BYTE;
	myDataLen		:__XINT:=75 * 3 + 16;
	
	init			:BOOL :=TRUE;	
	fmc				:findMasterCtrl;
	gs				:getStateByIdx;
END_VAR



//initialize
IF init THEN
	init := FALSE;
	tcpConnector(InetAddress := destIp,port:= destPort);
END_IF

prepareMetaData();

tcpConnector.send(dataLength := myDataLen, sendBuf := myData);

METHOD prepareMetaData
VAR_INPUT
END_VAR
VAR
	i0				:INT;
	i1				:INT;
	
	pos				:INT;
	
	intTmp			:UINT;
	byte1			:BYTE;
	byte2			:BYTE;
	plugStat		:BYTE;
	
	mCtrl			:INT;
END_VAR
VAR CONSTANT
	aOil	:ARRAY [1..7] OF INT :=[9,11,8,8,8,8,23];		
END_VAR
//data head (decimal)
myData[1]	:=	83	;
myData[2]	:=	70	;
myData[3]	:=	68	;
myData[4]	:=	84	;

//data length
myData[5]	:=	0	;
myData[6]	:=	225	;

//healthy data
myData[7]	:=	0	;
myData[8]	:=	11	;

//zero
myData[9]	:=	0	;
myData[10]	:=	0	;
myData[11]	:=	0	;
myData[12]	:=	0	;

myData[13]	:=	0	;
myData[14]	:=	0	;
myData[15]	:=	0	;
myData[16]	:=	0	;

//list
pos := 17;
FOR i0:=1 TO 7 DO
	FOR i1:=1 TO aOil[i0] DO
		intTmp := REAL_TO_UINT(gImple.PV_GroupTi.arrPV[i0].sNum[i1].posVal.Current * 10);
		
		//test
		//intTmp := INT_TO_UINT(800 + i1 * 10);
		
		
		byte1 := INT_TO_BYTE(SHR(intTmp, 8)); 
		byte2 := INT_TO_BYTE(intTmp AND 255); 
		fmc(grp := i0, num := i1, ctrl => mCtrl);
		gs(grp := i0, ctrl := mCtrl, state => plugStat);
		
		//test
		//byte3 := INT_TO_BYTE(i0 * 100 + i1);
		myData[pos] := plugStat;
		pos := pos + 1;		
		myData[pos] := byte1;
		pos := pos + 1;
		myData[pos] := byte2;
		pos := pos + 1;
		
		
	END_FOR
END_FOR
END_METHOD

END_PROGRAM

// Device/Application/dataUpload/tcpUpload
FUNCTION_BLOCK tcpUpload
VAR_INPUT
	InetAddress		:STRING;
	port			:UINT;
END_VAR
VAR_OUTPUT
END_VAR
VAR
	tcpConnector	:TCP.Connector;
	tcpStream		:TCP.Stream;
	pointerStream	:POINTER TO TCP.Stream;


	tcpState		:UINT:=0;
	tcpCount		:UINT:=0;
	
	netState		:INT;


END_VAR

METHOD send
VAR_INPUT
	
	dataLength		:__XINT;
	sendBuf 		:ARRAY[1..1024]OF BYTE;
END_VAR
VAR
	sizeData		:__XINT;
END_VAR

tcpCount := tcpCount + 1;

CASE tcpState OF

	0:			//connet server
		tcpConnector.Connect(sIPAddress:= InetAddress,uiPort:= 60000,pStream => pointerStream);
		IF pointerStream<>0 THEN
			tcpState :=1;
		ELSE
			tcpState :=2;
		END_IF
		
	1:			
		netState := pointerStream^.Send(ADR(sendBuf),dataLength,diSent=>sizeData);			
		IF netState <> 0 THEN
			tcpState := 2;	
		END_IF
		
		
	2:		 	//断开连接
	    tcpConnector.Disconnect();
		tcpState := 0;

END_CASE
END_METHOD

END_FUNCTION_BLOCK

// Device/Application/dataUpload/findMasterCtrl
FUNCTION_BLOCK findMasterCtrl
VAR_INPUT
	grp			:	INT;
	num			:	INT;
END_VAR
VAR_OUTPUT
	ctrl		:	INT;	

END_VAR
VAR
END_VAR

//已知比例阀组索引和油缸编号,获取对应开关阀索引
CASE grp OF
	1:
		CASE num OF
			1:		ctrl := 1;
			2:		ctrl := 1;
			3:		ctrl := 2;
			4:		ctrl := 2;
			5:		ctrl := 3;
			6:		ctrl := 4;
			7:		ctrl := 4;
			8:		ctrl := 5;
			9:		ctrl := 6;
			ELSE	ctrl := -1;
		END_CASE

	2:
		CASE num OF
			1:		ctrl := 1;
			2:		ctrl := 1;
			3:		ctrl := 1;
			4:		ctrl := 2;
			5:		ctrl := 3;
			6:		ctrl := 3;
			7:		ctrl := 3;
			8:		ctrl := 4;
			9:		ctrl := 5;
			10:		ctrl := 5;
			11:		ctrl := 5;
			ELSE	ctrl := -1;
		END_CASE

	3:
		CASE num OF
			1:		ctrl := 1;
			2:		ctrl := 1;
			3:		ctrl := 1;
			4:		ctrl := 1;
			5:		ctrl := 1;
			6:		ctrl := 1;
			7:		ctrl := 1;
			8:		ctrl := 1;
			ELSE	ctrl := -1;
		END_CASE

	4:
		CASE num OF
			1:		ctrl := 1;
			2:		ctrl := 1;
			3:		ctrl := 1;
			4:		ctrl := 1;
			5:		ctrl := 1;
			6:		ctrl := 1;
			7:		ctrl := 1;
			8:		ctrl := 1;
			ELSE	ctrl := -1;
		END_CASE

	5:
		CASE num OF
			1:		ctrl := 1;
			2:		ctrl := 1;
			3:		ctrl := 1;
			4:		ctrl := 1;
			5:		ctrl := 1;
			6:		ctrl := 1;
			7:		ctrl := 1;
			8:		ctrl := 1;
			ELSE	ctrl := -1;
		END_CASE
		
		
	6:
		CASE num OF
			1:		ctrl := 1;
			2:		ctrl := 1;
			3:		ctrl := 2;
			4:		ctrl := 3;
			5:		ctrl := 3;
			6:		ctrl := 4;
			7:		ctrl := 5;
			8:		ctrl := 5;
			ELSE	ctrl := -1;
		END_CASE

	7:
		CASE num OF
			1:		ctrl := 1;
			2:		ctrl := 1;
			3:		ctrl := 1;
			4:		ctrl := 1;
			5:		ctrl := 2;
			6:		ctrl := 3;
			7:		ctrl := 3;
			8:		ctrl := 3;
			9:		ctrl := 3;
			10:		ctrl := 4;
			11:		ctrl := 4;
			12:		ctrl := 4;
			13:		ctrl := 4;
			14:		ctrl := 4;
			15:		ctrl := 5;
			16:		ctrl := 5;
			17:		ctrl := 5;
			18:		ctrl := 5;
			19:		ctrl := 5;
			20:		ctrl := 6;
			21:		ctrl := 6;
			22:		ctrl := 7;
			23:		ctrl := 7;
			ELSE	ctrl := -1;
		END_CASE


	ELSE
		ctrl := -1;
		
END_CASE

END_FUNCTION_BLOCK

// Device/Application/dataUpload/getStateByIdx
FUNCTION_BLOCK getStateByIdx
VAR_INPUT
	grp			:	INT;
	ctrl		:	INT;
END_VAR
VAR_OUTPUT
	state		:	BYTE;
END_VAR
VAR
END_VAR


CASE gImple.PV_GroupTi.arrPV[grp].sColumn[ctrl].eStat OF
	cmdStat.eNormal:
		state := 0;
	cmdStat.eRun:
		state := 1;
	cmdStat.Extend_Done:
		state := 2;
	cmdStat.Retract_Done:
		state := 3;
	cmdStat.eError:
		state := 4;
	ELSE
		state := 0;

END_CASE

END_FUNCTION_BLOCK

// Device/Application/can/canTx
PROGRAM canTx
VAR
		T_CNT   :UINT;

END_VAR

T_CNT := T_CNT+1;
IF  T_CNT > 1000 THEN
	 T_CNT := 1;
END_IF


swmc_C05_Tx(T_CNT,ADR(gImple.PV_GroupTi));
swmc_C06_Tx(T_CNT,ADR(gImple.PV_GroupTi));

END_PROGRAM

// Device/Application/can/swmc_C05_Tx
FUNCTION swmc_C05_Tx : BOOL
VAR_INPUT
	CNT				: UINT;
	psPVTi			: POINTER TO propValveModule_Ti;
END_VAR
VAR
	senddata	: ARRAY[1..8] OF BYTE;
	Send_cnt	: UINT;
END_VAR

//控制速度--待定
Send_cnt :=  CNT MOD 5;

CASE Send_cnt OF
	
    1:
	 //C1-0x450
	senddata[1] :=  WORD_TO_BYTE(psPVTi^.arrPV[1].percenVal);  		   //发送DTE1比例阀值
	senddata[2] :=  WORD_TO_BYTE(SHR(psPVTi^.arrPV[1].percenVal,8));     
	senddata[3] :=  WORD_TO_BYTE(psPVTi^.arrPV[2].percenVal);  		   //发送DTE2比例阀值
	senddata[4] :=  WORD_TO_BYTE(SHR(psPVTi^.arrPV[2].percenVal,8));   
	senddata[5] :=  WORD_TO_BYTE(psPVTi^.arrPV[3].percenVal);  		   //发送DTE3比例阀值
	senddata[6] :=  WORD_TO_BYTE(SHR(psPVTi^.arrPV[3].percenVal,8));     
	senddata[7] :=  WORD_TO_BYTE(psPVTi^.arrPV[4].percenVal);  		   //发送DTE4比例阀值
	senddata[8] :=  WORD_TO_BYTE(SHR(psPVTi^.arrPV[4].percenVal,8));    //0-65535  对应0-100  
	//发送至C5
	CAN_Send_Data_SWMC(5, 16#450,senddata);   //发送ID 0x450到C5
	
	2:
	 //C5-0x451
	senddata[1] :=  WORD_TO_BYTE(psPVTi^.arrPV[5].percenVal);  		   //发送DTE5比例阀值
	senddata[2] :=  WORD_TO_BYTE(SHR(psPVTi^.arrPV[5].percenVal,8));    //0-65535  对应0-100  
	
	senddata[3].0:=  psPVTi^.arrPV[1].sColumn[1].bE_Open;
	senddata[3].1:=  psPVTi^.arrPV[1].sColumn[1].bR_Open;  
//***************** 
    senddata[3].4:=  psPVTi^.arrPV[1].sColumn[2].bE_Open;
	senddata[3].5:=  psPVTi^.arrPV[1].sColumn[2].bR_Open; 
//******************
	senddata[3].2:=  psPVTi^.arrAddtion[2].sPlateCtrl.bExtend;
	senddata[3].3:=  psPVTi^.arrAddtion[2].sPlateCtrl.bRetract;
//*****************  
	senddata[4].0:=  psPVTi^.arrPV[1].sColumn[6].bE_Open;               
	senddata[4].1:=  psPVTi^.arrPV[1].sColumn[6].bR_Open;			
	senddata[4].2:=  psPVTi^.arrPV[1].sColumn[4].bE_Open;               
	senddata[4].3:=  psPVTi^.arrPV[1].sColumn[4].bR_Open;		
	
	senddata[5].0:=  psPVTi^.arrPV[1].sColumn[5].bE_Open;               
	senddata[5].1:=  psPVTi^.arrPV[1].sColumn[5].bR_Open;          
	senddata[5].2:=  psPVTi^.arrPV[1].sColumn[3].bE_Open;               
	senddata[5].3:=  psPVTi^.arrPV[1].sColumn[3].bR_Open;         
	
	senddata[6].0:=  psPVTi^.arrPV[2].sColumn[1].bE_Open;               
	senddata[6].1:=  psPVTi^.arrPV[2].sColumn[1].bR_Open;          
	//发送至C5
	CAN_Send_Data_SWMC(5, 16#451,senddata);				//发送ID 0x451到C5
	
	3:
	 //C5.1 IO-0x452
	senddata[1].0:=  psPVTi^.arrPV[2].sColumn[2].bE_Open;               
	senddata[1].1:=  psPVTi^.arrPV[2].sColumn[2].bR_Open;       
	
	senddata[2].0:=  psPVTi^.arrPV[2].sColumn[3].bE_Open;               
	senddata[2].1:=  psPVTi^.arrPV[2].sColumn[3].bR_Open; 	       

	senddata[3].0:=  psPVTi^.arrPV[2].sColumn[4].bE_Open;               
	senddata[3].1:=  psPVTi^.arrPV[2].sColumn[4].bR_Open;			
		
	senddata[4].0:=  psPVTi^.arrPV[2].sColumn[5].bE_Open;               
	senddata[4].1:=  psPVTi^.arrPV[2].sColumn[5].bR_Open;			
	//发送至C5
	CAN_Send_Data_SWMC(5, 16#452,senddata);				//发送ID 0x452到C5.1
	
	4:
	 //C5.2 IO-0x453
	senddata[1].0:=  psPVTi^.arrPV[3].sColumn[1].bE_Open;               
	senddata[1].1:=  psPVTi^.arrPV[3].sColumn[1].bR_Open;         
	
	senddata[2].0:=  psPVTi^.arrPV[4].sColumn[1].bE_Open;               
	senddata[2].1:=  psPVTi^.arrPV[4].sColumn[1].bR_Open; 	      
	
	senddata[3].0:=  psPVTi^.arrPV[5].sColumn[1].bE_Open;               
	senddata[3].1:=  psPVTi^.arrPV[5].sColumn[1].bR_Open;			
	//发送至C5
	CAN_Send_Data_SWMC(5, 16#453,senddata);				//发送ID 0x453到C5.2

END_CASE

END_FUNCTION

// Device/Application/can/CAN_Send_Data_SWMC
FUNCTION CAN_Send_Data_SWMC : BOOL
VAR_INPUT
	SWMC_ID : UINT;
	id 		: UINT;
	data	: ARRAY[1..8] OF BYTE;
END_VAR
VAR
	
END_VAR

CASE  SWMC_ID OF

	5:
		gCan.C5TxMsg.TXMsg[1].TxMsg_CobId 	:= 8 + 32 * id;
	  	gCan.C5TxMsg.TXMsg[1].TxMsg_Byte 	:= data;
	   	gCan.C5TxMsg.NoOfTxMessages			:= 1;
	   	gCan.C5TxMsg.TxCounter 				:= gCan.C5TxMsg.TxCounter +1;
	
	6:
		gCan.C6TxMsg.TXMsg[1].TxMsg_CobId 	:= 8 + 32 * id;
	  	gCan.C6TxMsg.TXMsg[1].TxMsg_Byte 	:= data;
	   	gCan.C6TxMsg.NoOfTxMessages			:= 1;
	   	gCan.C6TxMsg.TxCounter 				:= gCan.C6TxMsg.TxCounter +1;
	

END_CASE

END_FUNCTION

// Device/Application/can/swmc_C06_Tx
FUNCTION swmc_C06_Tx : BOOL
VAR_INPUT
	CNT				: UINT;
	psPVTi			: POINTER TO propValveModule_Ti;
END_VAR
VAR
	senddata	: ARRAY[1..8] OF BYTE;
	Send_cnt	: UINT;
END_VAR

//控制速度--待定
Send_cnt :=  CNT MOD 5;

CASE Send_cnt OF
	
    1:
	 //C6-0x460
	senddata[1] :=  WORD_TO_BYTE(psPVTi^.arrPV[6].percenVal);  		   //发送DTE6比例阀值
	senddata[2] :=  WORD_TO_BYTE(SHR(psPVTi^.arrPV[6].percenVal,8));     
	senddata[3] :=  WORD_TO_BYTE(psPVTi^.arrPV[7].percenVal);  		   //发送DTE7比例阀值
	senddata[4] :=  WORD_TO_BYTE(SHR(psPVTi^.arrPV[7].percenVal,8));   
	
	senddata[5].0:=  psPVTi^.arrPV[6].sColumn[1].bE_Open;               
	senddata[5].1:=  psPVTi^.arrPV[6].sColumn[1].bR_Open;          
	senddata[5].2:=  psPVTi^.arrPV[6].sColumn[2].bE_Open;               
	senddata[5].3:=  psPVTi^.arrPV[6].sColumn[2].bR_Open;         

	senddata[6].0:=  psPVTi^.arrPV[6].sColumn[3].bE_Open;               
	senddata[6].1:=  psPVTi^.arrPV[6].sColumn[3].bR_Open;          
	senddata[6].2:=  psPVTi^.arrPV[6].sColumn[4].bE_Open;               
	senddata[6].3:=  psPVTi^.arrPV[6].sColumn[4].bR_Open;         
	senddata[6].4:=  psPVTi^.arrAddtion[1].sPlateCtrl.bExtend;
	senddata[6].5:=  psPVTi^.arrAddtion[1].sPlateCtrl.bRetract;
	
	senddata[7].0:=  psPVTi^.arrPV[6].sColumn[5].bE_Open;               
	senddata[7].1:=  psPVTi^.arrPV[6].sColumn[5].bR_Open;          
	senddata[7].2:=  psPVTi^.arrPV[7].sColumn[1].bE_Open;               
	senddata[7].3:=  psPVTi^.arrPV[7].sColumn[1].bR_Open;         

	senddata[8].0:=  psPVTi^.arrPV[7].sColumn[2].bE_Open;               
	senddata[8].1:=  psPVTi^.arrPV[7].sColumn[2].bR_Open;          
	senddata[8].2:=  psPVTi^.arrPV[7].sColumn[3].bE_Open;               
	senddata[8].3:=  psPVTi^.arrPV[7].sColumn[3].bR_Open;         

	//发送至C6
	CAN_Send_Data_SWMC(6, 16#460,senddata);   //发送ID 0x460到C6
	
	2:
	 //C6.1 IO-0x461
	senddata[1].0:=  psPVTi^.arrPV[7].sColumn[4].bE_Open;  		
	senddata[1].1:=  psPVTi^.arrPV[7].sColumn[4].bR_Open;   	
	
	senddata[2].0:=  psPVTi^.arrPV[7].sColumn[5].bE_Open;
	senddata[2].1:=  psPVTi^.arrPV[7].sColumn[5].bR_Open;   
  
	senddata[3].0:=  psPVTi^.arrPV[7].sColumn[6].bE_Open;               
	senddata[3].1:=  psPVTi^.arrPV[7].sColumn[6].bR_Open;			

	senddata[4].0:=  psPVTi^.arrPV[7].sColumn[7].bE_Open;               
	senddata[4].1:=  psPVTi^.arrPV[7].sColumn[7].bR_Open;          
    
	//发送至C6
	CAN_Send_Data_SWMC(6, 16#461,senddata);				//发送ID 0x461到C6
	
END_CASE

END_FUNCTION

// Device/Application/modbus/modbusAct
PROGRAM modbusAct
VAR
	bInitialize				:BOOL:=TRUE;
	iClientConnect			:UINT;
	iCountAct				:UINT:=10;
	iTemp					:UINT;
	iErrCode				:BYTE;

	fbModbusClient				: ModbusTcp_Client;
	fbReadHoldRegister  		: ReadHoldRegister;					//读保持寄存器
	fbWriteSingleHoldRegister	: WriteSingleHoldRegister;			//写保持1寄存器

	fbWriteMutiRegister			: WriteMutiRegister;	
	fbLogSav					: logSave;

END_VAR

IF bInitialize THEN
	initAddrPacket(ADR(gModbus.master));
	bInitialize:=FALSE;
END_IF

IF iClientConnect<>1 THEN
	//fbModbusClient(sIPAddress:='192.168.2.23',uiPort:=520);//连接IPC
	fbModbusClient(sIPAddress:='192.168.5.55',uiPort:=502);//连接工控机
END_IF

IF fbModbusClient.bSuccess THEN
	iClientConnect:=1;

	CASE iCountAct OF
	
		10:
			modbusAct.handleToken();
		20:
			modbusAct.handleCommand1();//平台指令接收
		30:			
			modbusAct.handleStatus1();//发送到位指令
	
	END_CASE

END_IF

METHOD PRIVATE initAddrPacket : BOOL
VAR_INPUT
	pModbus			: POINTER TO ModbusStructx;
END_VAR

pModbus^.sCmd.wStartAddr		:= 10;
pModbus^.sCmd.wAmount			:= 6;

pModbus^.sStatus.wStartAddr		:= 110;
pModbus^.sStatus.wAmount		:= 96;

pModbus^.sToken.wStartAddr		:=42;
pModbus^.sToken.wAmount			:=1;
END_METHOD

ACTION handleToken:
fbReadHoldRegister(
	xExecute	:=TRUE,
	slaveId		:=1,
	wStartAdr	:=gModbus.master.sToken.wStartAddr,
	wLen		:=gModbus.master.sToken.wAmount,
	pTcpStream	:= fbModbusClient.pfbTcpStream,
	modbusHoldRegData:= gModbus.arrBufferDat);

IF fbReadHoldRegister.bSucced THEN

	gModbus.master.sToken.iNo:=gModbus.arrBufferDat[gModbus.master.sToken.wStartAddr];
	fbReadHoldRegister(
		xExecute := FALSE,
		modbusHoldRegData:=g_modbusHoldRegData);

	iCountAct :=20;		

END_IF

IF fbReadHoldRegister.berror THEN
	fbReadHoldRegister(
		xExecute :=FALSE,
	modbusHoldRegData:= gModbus.arrBufferDat);
	fbModbusClient.M_Reset();
	iClientConnect :=0;
	iCountAct:=10;	
	iErrCode:=fbReadHoldRegister.errCode;
END_IF
END_ACTION

ACTION handleCommand1:
fbReadHoldRegister(
	xExecute	:= TRUE,
	slaveId		:= 1,
	wStartAdr	:= 10,
	wLen		:= 48,
	pTcpStream	:= fbModbusClient.pfbTcpStream,
	modbusHoldRegData:= gModbus.arrBufferDat);

IF fbReadHoldRegister.bSucced THEN
	FOR iTemp:=0 TO 5 DO
		gModbus.master.sCmd.arrDat[10+iTemp] := gModbus.arrBufferDat[gModbus.master.sCmd.wStartAddr+iTemp];	
	END_FOR
	gModbus.master.sCmd.arrDat[49] := gModbus.arrBufferDat[49];	
	fbReadHoldRegister(
		xExecute := FALSE,
		modbusHoldRegData:=g_modbusHoldRegData);
	modbusAct.executeCmd();

	iCountAct :=30;		
END_IF

IF fbReadHoldRegister.berror THEN
	fbReadHoldRegister(
		xExecute :=FALSE,
		modbusHoldRegData:= gModbus.arrBufferDat);
	fbModbusClient.M_Reset();
	iClientConnect :=0;
	iCountAct:=10;	
	iErrCode:=fbReadHoldRegister.errCode;
END_IF
END_ACTION

ACTION handleStatus1:

modbusAct.getStatus();	//获取位置

fbWriteMutiRegister(
	xExecute	:= TRUE,
	slaveId		:= 1,
	startAddr	:= 110,			//110-205
	wRegNum		:= 96, //gModbus.master.sStatus.wAmount
	value		:= ADR(gModbus.master.sStatus.arrDat),
	pTcpStream	:= fbModbusClient.pfbTcpStream);
	
IF fbWriteMutiRegister.bSucced THEN
	fbWriteMutiRegister(xExecute:=FALSE);
	iCountAct:=10;
END_IF

IF fbWriteMutiRegister.berror THEN
	fbWriteMutiRegister(xExecute:=FALSE);
	fbModbusClient.M_Reset();
	iCountAct:=10;
	iClientConnect:=0;
	iErrCode :=fbWriteMutiRegister.errCode;
END_IF
END_ACTION

METHOD  PRIVATE executeCmd 
VAR_INPUT
END_VAR
VAR 
	bToken				:BOOL;
	iTemp1				:USINT;
	iTemp2				:USINT;
	fbGetObjCmdIndex	:getObjIndexC;
	fbgetCol			:getColumnStr;
	iN1					:USINT;
	iN2					:USINT;
	strLogW				:STRING;
	strLogOut			:STRING;

	
END_VAR
//检测是否为同一指令
(*gModbus.master.sToken.iNew:=gModbus.master.sToken.iNo;
IF gModbus.master.sToken.iLast<>gModbus.master.sToken.iNew THEN
	gModbus.master.sToken.iLast:=gModbus.master.sToken.iNew;
	bToken:=TRUE;
ELSE
	bToken:=FALSE;
END_IF

IF bToken THEN*)
	
FOR iTemp:=10 TO 15 DO
	gModbus.master.sCmd.arrNew[iTemp,0]:=gModbus.master.sCmd.arrDat[iTemp].0;
	gModbus.master.sCmd.arrNew[iTemp,1]:=gModbus.master.sCmd.arrDat[iTemp].1;
	gModbus.master.sCmd.arrNew[iTemp,2]:=gModbus.master.sCmd.arrDat[iTemp].2;
	gModbus.master.sCmd.arrNew[iTemp,3]:=gModbus.master.sCmd.arrDat[iTemp].3;
	gModbus.master.sCmd.arrNew[iTemp,4]:=gModbus.master.sCmd.arrDat[iTemp].4;
	gModbus.master.sCmd.arrNew[iTemp,5]:=gModbus.master.sCmd.arrDat[iTemp].5;
	gModbus.master.sCmd.arrNew[iTemp,6]:=gModbus.master.sCmd.arrDat[iTemp].6;
	gModbus.master.sCmd.arrNew[iTemp,7]:=gModbus.master.sCmd.arrDat[iTemp].7;
	gModbus.master.sCmd.arrNew[iTemp,8]:=gModbus.master.sCmd.arrDat[iTemp].8;
	gModbus.master.sCmd.arrNew[iTemp,9]:=gModbus.master.sCmd.arrDat[iTemp].9;
	gModbus.master.sCmd.arrNew[iTemp,10]:=gModbus.master.sCmd.arrDat[iTemp].10;
	gModbus.master.sCmd.arrNew[iTemp,11]:=gModbus.master.sCmd.arrDat[iTemp].11;
	gModbus.master.sCmd.arrNew[iTemp,12]:=gModbus.master.sCmd.arrDat[iTemp].12;
	gModbus.master.sCmd.arrNew[iTemp,13]:=gModbus.master.sCmd.arrDat[iTemp].13;
	gModbus.master.sCmd.arrNew[iTemp,14]:=gModbus.master.sCmd.arrDat[iTemp].14;
	gModbus.master.sCmd.arrNew[iTemp,15]:=gModbus.master.sCmd.arrDat[iTemp].15;
END_FOR	
	

FOR iTemp1:=10 TO 15 DO
	FOR iTemp2:=0 TO 15 DO
		IF gModbus.master.sCmd.arrNew[iTemp1,iTemp2]<>gModbus.master.sCmd.arrLast[iTemp1,iTemp2] THEN	//上升沿检测
		IF gModbus.master.sCmd.arrNew[iTemp1,iTemp2]=TRUE THEN
			fbGetObjCmdIndex(iAdr:=iTemp1,iBit:=iTemp2,iO1=>iN1,iO2=>iN2);
			//fbgetCol(iI1:=iN1,iI2:=iN2,strO=>strLogW);
			IF iN1<>0 AND iN2<>0 THEN
				IF iTemp1<13 THEN
					gUI.TiG.arrPV[iN1].sColumn[iN2].bExtend:=TRUE;
					//strLogW:=concat(strLogW,'->extern');
				ELSE
					gUI.TiG.arrPV[iN1].sColumn[iN2].bRetract:=TRUE;
					//strLogW:=concat(strLogW,'->retract');
				END_IF
				//fbLogSav(Log_Data:= strLogW, FilePath:= 'D:/log', Name_Flag:= 'skyRail', cycle:= T#60S, Out_log=> strLogOut);
			END_IF
		END_IF	
		END_IF
	END_FOR	
END_FOR
(*
IF gModbus.master.sCmd.arrNew[10,12]<>gModbus.master.sCmd.arrLast[10,12] THEN
IF gModbus.master.sCmd.arrNew[10,12]=TRUE THEN
	gUI.TiG.arrPlate[1].sCmd.bExtend:=TRUE;gUI.TiG.arrPlate[1].sCmd.bRetract:=FALSE;
	//fbLogSav(Log_Data:= 'Plate1->extern', FilePath:= 'D:/log', Name_Flag:= 'skyRail', cycle:= T#60S, Out_log=> strLogOut);
END_IF	
END_IF
IF gModbus.master.sCmd.arrNew[10,13]<>gModbus.master.sCmd.arrLast[10,13] THEN
IF gModbus.master.sCmd.arrNew[10,13]=TRUE THEN
	gUI.TiG.arrPlate[2].sCmd.bExtend:=TRUE;gUI.TiG.arrPlate[2].sCmd.bRetract:=FALSE;
	//fbLogSav(Log_Data:= 'Plate2->extern', FilePath:= 'D:/log', Name_Flag:= 'skyRail', cycle:= T#60S, Out_log=> strLogOut);
END_IF	
END_IF
IF gModbus.master.sCmd.arrNew[13,12]<>gModbus.master.sCmd.arrLast[13,12] THEN
IF gModbus.master.sCmd.arrNew[13,12]=TRUE THEN
	gUI.TiG.arrPlate[1].sCmd.bExtend:=FALSE;gUI.TiG.arrPlate[1].sCmd.bRetract:=TRUE;
	//fbLogSav(Log_Data:= 'Plate1->retract', FilePath:= 'D:/log', Name_Flag:= 'skyRail', cycle:= T#60S, Out_log=> strLogOut);
END_IF	
END_IF
IF gModbus.master.sCmd.arrNew[13,13]<>gModbus.master.sCmd.arrLast[13,13] THEN
IF gModbus.master.sCmd.arrNew[13,13]=TRUE THEN
	gUI.TiG.arrPlate[2].sCmd.bExtend:=FALSE;gUI.TiG.arrPlate[2].sCmd.bRetract:=TRUE;
	//fbLogSav(Log_Data:= 'Plate2->retract', FilePath:= 'D:/log', Name_Flag:= 'skyRail', cycle:= T#60S, Out_log=> strLogOut);
END_IF	
END_IF

FOR iTemp1:=10 TO 15 DO
	FOR iTemp2:=0 TO 15 DO
		gModbus.master.sCmd.arrLast[iTemp1,iTemp2]:=gModbus.master.sCmd.arrNew[iTemp1,iTemp2];	
	END_FOR		
END_FOR	
*)	
	
//END_IF
END_METHOD

METHOD PRIVATE getStatus : BOOL
VAR_INPUT
	
END_VAR
VAR
	iVT					:INT;
	iVT1				:INT;
	iOAde				:USINT;	
	iOAdr				:USINT;	
	fbNumMapE			:getObjIndexE;
	fbNumMapR			:getObjIndexR;
	
END_VAR
VAR CONSTANT
	aNo		:ARRAY [1..7] OF INT :=[6, 5,1,1,1,5, 7];		//每个比例阀下开关阀的数量(天轨):arrMappingRealNumTiG
END_VAR

FOR iVT:=1 TO 7 DO				//每个比例阀
	FOR iVT1:=1 TO aNo[iVT] DO	//比例阀中每个开关阀
		fbNumMapE(iI1:=iVT,iI2:=iVT1,iAdr=>iOAde);
		fbNumMapR(iI1:=iVT,iI2:=iVT1,iAdr=>iOAdr);	
		IF gImple.PV_GroupTi.arrPV[iVT].sColumn[iVT1].eStat=cmdStat.Extend_Done THEN
			gModbus.master.sStatus.arrDat[iOAde]:=1;
		ELSE
			gModbus.master.sStatus.arrDat[iOAde]:=0;
		END_IF
		IF gImple.PV_GroupTi.arrPV[iVT].sColumn[iVT1].eStat=cmdStat.Retract_Done THEN
			gModbus.master.sStatus.arrDat[iOAdr]:=1;
		ELSE
			gModbus.master.sStatus.arrDat[iOAdr]:=0;
		END_IF		

	END_FOR	
END_FOR


(*
IF gImple.PV_GroupTi.arrAddtion[1].sPlateStatus.eStat=cmdStat.Extend_Done THEN
	gModbus.master.sStatus.arrDat[122]:=1;
ELSE
	gModbus.master.sStatus.arrDat[122]:=0;	
END_IF
IF gImple.PV_GroupTi.arrAddtion[1].sPlateStatus.eStat=cmdStat.Retract_Done THEN
	gModbus.master.sStatus.arrDat[153]:=1;
ELSE
	gModbus.master.sStatus.arrDat[153]:=0;	
END_IF

IF gImple.PV_GroupTi.arrAddtion[2].sPlateStatus.eStat=cmdStat.Extend_Done THEN
	gModbus.master.sStatus.arrDat[123]:=1;
ELSE
	gModbus.master.sStatus.arrDat[123]:=0;	
END_IF
IF gImple.PV_GroupTi.arrAddtion[2].sPlateStatus.eStat=cmdStat.Retract_Done THEN
	gModbus.master.sStatus.arrDat[154]:=1;
ELSE
	gModbus.master.sStatus.arrDat[153]:=0;	
END_IF
*)

//gModbus.master.sStatus.arrDat[]:=xx;
//gImple.PV_GroupTi.arrPV[iVT].sColumn[iVT1].eStat:=cmdStat.Extend_Done;
END_METHOD

END_PROGRAM

// Device/Application/public_datum/datarecord/logSave
FUNCTION_BLOCK logSave
VAR_INPUT
	Log_Data	: STRING;					// 数据输入 一次最大可以写入200个数据
	FilePath 	: STRING := 'C:/DataSave'; 	// 存储文件夹
	Name_Flag	: STRING := 'Log';			// 文件标志
	cycle		: TIME;						// 更新一个文件夹时间
END_VAR
VAR_OUTPUT
	Out_log		:STRING;
END_VAR
VAR
	datetime	: DATE_AND_TIME;
	uiYear 		: UINT; 
    uiMonth 	: UINT; 
    uiDay 		: UINT; 
    uiHour 		: UINT; 
    uiMinute 	: UINT; 
    uiSecond 	: UINT;	
	uiMsSecond	: UINT;
	Last_S		: UINT:=100;
	UdMsOffset  : UDINT;
	UdIntms 	: UDINT;
	DTimer_Str  : STRING;
END_VAR
VAR
	File_Init	: BOOL :=TRUE;
	Log_t_Init :BOOL:=TRUE;
	New_File_Ton: TON;
	Filename	: STRING;
	F_HANDL		: DWORD;
	F_err		: DWORD;
	F_pos		: DWORD;
	log_Str		: STRING;
END_VAR

datetime:=GetDateTime();   //获取时间
DTU.DTSplit(
		dtDateAndTime:= datetime, 
		puiYear:= ADR(uiYear), 
		puiMonth:=  ADR(uiMonth), 
		puiDay:=  ADR(uiDay), 
		puiHour:=  ADR(uiHour), 
		puiMinute:=  ADR(uiMinute), 
		puiSecond:= ADR(uiSecond) );

IF  Log_t_Init THEN			//日志时间初始化
	IF uiSecond = Last_S +1 OR  uiSecond = Last_S -59 THEN
		UdMsOffset := SysTimeGetMs();
		Last_S :=  uiSecond;
	ELSE
		Last_S :=  uiSecond;
		RETURN;
	END_IF
    Log_t_Init := FALSE;
END_IF

IF 	File_Init  THEN          //创建文件
	Filename := FilePath;
	Filename := concat(Filename,'/');
	Filename := concat(Filename,Name_Flag);
	Filename := concat(Filename,UINT_TO_STRING(uiYear));
	Filename := concat(Filename,'_');
	Filename := concat(Filename,UINT_TO_STRING(uiMonth));
	Filename := concat(Filename,'_');
	Filename := concat(Filename,UINT_TO_STRING(uiDay));
	Filename := concat(Filename,'_');
	Filename := concat(Filename,UINT_TO_STRING(uiHour+8));
 	Filename := concat(Filename,'_');
	Filename := concat(Filename,UINT_TO_STRING(uiMinute));
	Filename := concat(Filename,'_');
	Filename := concat(Filename,UINT_TO_STRING(uiSecond));
    Filename := concat(Filename,'_log.log');
	F_HANDL :=SysFileOpen(szFile:= Filename, am:=ACCESS_MODE.AM_WRITE, pResult:= ADR(F_err));  //创建新文件
	SysFileClose(hFile:=F_HANDL );
	File_Init := FALSE;
	New_File_Ton(IN:= FALSE , PT:= cycle, Q=> , ET=> );  //复位
END_IF

New_File_Ton(IN:= TRUE , PT:= cycle, Q=> , ET=> );			//小时创建一个新文件
IF New_File_Ton.Q THEN
	File_Init := TRUE;	
END_IF

UdIntms := SysTimeGetMs();
uiMsSecond := UDINT_TO_UINT((UdIntms - UdMsOffset)MOD 1000);   //计算微秒
DTimer_Str := UINT_TO_STRING(uiYear);
DTimer_Str := concat(DTimer_Str,'-');
DTimer_Str := concat(DTimer_Str,UINT_TO_STRING(uiMonth));
DTimer_Str := concat(DTimer_Str,'-');
DTimer_Str := concat(DTimer_Str,UINT_TO_STRING(uiDay));
DTimer_Str := concat(DTimer_Str,' ');
DTimer_Str := concat(DTimer_Str,UINT_TO_STRING(uiHour+8));
DTimer_Str := concat(DTimer_Str,':');
DTimer_Str := concat(DTimer_Str,UINT_TO_STRING(uiMinute));
DTimer_Str := concat(DTimer_Str,':');
DTimer_Str := concat(DTimer_Str,UINT_TO_STRING(uiSecond));
DTimer_Str := concat(DTimer_Str,':');
DTimer_Str := concat(DTimer_Str,UINT_TO_STRING(uiMsSecond));
DTimer_Str := concat(DTimer_Str,'    ');

log_Str := concat(Log_Data,'$R');
F_HANDL :=SysFileOpen(szFile:= Filename, am:=ACCESS_MODE.AM_APPEND, pResult:= ADR(F_err));  //打开文件
SysFileGetPos(hFile:= F_HANDL , pulPos:= ADR(F_pos));		//获取文件位置
SysFileSetPos(hFile:= F_HANDL, ulOffset:= F_pos);
SysFileWrite(hFile:=F_HANDL , pbyBuffer:= ADR(DTimer_Str) , ulSize:= SysStrLen(DTimer_Str) , pResult:= ADR(F_err));		// 写入时间
SysFileWrite(hFile:=F_HANDL , pbyBuffer:= ADR(log_Str) , ulSize:= SysStrLen(log_Str) , pResult:= ADR(F_err));		// 写入数据
SysFileClose(hFile:=F_HANDL );

Out_log := concat(DTimer_Str,log_Str);

END_FUNCTION_BLOCK

// Device/Application/modbus/getObjIndexC
FUNCTION_BLOCK FINAL getObjIndexC
VAR_INPUT
	iAdr	:UINT;
	iBit	:UINT;
END_VAR
VAR_OUTPUT
	iO1		:USINT;
	iO2		:USINT;
END_VAR
VAR
END_VAR

//已知指令地址，获取对应比例阀索引及油缸编号索引
CASE iAdr OF
	10,13:
		CASE iBit OF
			1:		iO1:=3;iO2:=1;//Q01-04
			2:		iO1:=4;iO2:=1;//Q05-08
			3:		iO1:=5;iO2:=1;//Q09-12
			4:		iO1:=6;iO2:=1;//Q13-14
			5:		iO1:=6;iO2:=2;//Q15
			6:		iO1:=7;iO2:=4;//Q17-21
			7:		iO1:=7;iO2:=5;//Q22-26
			8:		iO1:=1;iO2:=5;//Q28
			9:		iO1:=1;iO2:=4;//Q29-30
			ELSE	iO1:=0;iO2:=0;	
		END_CASE

	11,14:
		CASE iBit OF
			0:		iO1:=1;iO2:=3;//L00
			ELSE	iO1:=0;iO2:=0;
		END_CASE	
	
	12,15:
		CASE iBit OF
			0:		iO1:=1;iO2:=6;//L01
			1:		iO1:=2;iO2:=1;//L02-04
			2:		iO1:=2;iO2:=2;//L05
			3:		iO1:=2;iO2:=3;//L06-08
			4:		iO1:=2;iO2:=4;//L09
			5:		iO1:=2;iO2:=5;//L10-12
			6:		iO1:=6;iO2:=4;//L13
			7:		iO1:=6;iO2:=3;//L14-15
			8:		iO1:=6;iO2:=5;//L16
			9:		iO1:=7;iO2:=6;//L17
			10:		iO1:=7;iO2:=1;//L18-21
			11:		iO1:=7;iO2:=2;//L22
			12:		iO1:=7;iO2:=3;//L23-26
			13:		iO1:=7;iO2:=7;//L27
			14:		iO1:=1;iO2:=1;//L28
			15:		iO1:=1;iO2:=2;//L29-30
			ELSE	iO1:=0;iO2:=0;
		END_CASE	
	ELSE
		iO1:=0;iO2:=0;	
END_CASE

END_FUNCTION_BLOCK

// Device/Application/modbus/getColumnStr
FUNCTION_BLOCK FINAL getColumnStr
VAR_INPUT
	iI1		:UINT;
	iI2		:UINT;
END_VAR
VAR_OUTPUT
	strO	:STRING;
END_VAR
VAR
END_VAR

CASE iI1 OF
	1:
	CASE iI2 OF
		1:strO:='E28L1-E28L2';
		2:strO:='E29L-E30L';
		3:strO:='E00L';
		4:strO:='E29Q-E30Q';
		5:strO:='E28Q';
		6:strO:='E01L';
	END_CASE
	2:
	CASE iI2 OF
		1:strO:='E02L-E04L';
		2:strO:='E05L';
		3:strO:='E06L-E08L';
		4:strO:='E09L';
		5:strO:='E10L-E12L';
	END_CASE
	3:strO:='E01Q1-E04Q2';
	4:strO:='E05Q1-E08Q2';
	5:strO:='E09Q1-E12Q2';
	6:
	CASE iI2 OF
		1:strO:='E13Q-E14Q';
		2:strO:='E15Q';
		3:strO:='E14L-E15L';
		4:strO:='E13L';
		5:strO:='E16L1-E16L2';

	END_CASE
	7:
	CASE iI2 OF
		1:strO:='E18L-E21L';
		2:strO:='E22L';
		3:strO:='E23L-E26L';
		4:strO:='E17Q-E21Q';
		5:strO:='E22Q-E26Q';
		6:strO:='E17L1-E17L2';
		7:strO:='E27L1-E27L2';
	END_CASE	
END_CASE

END_FUNCTION_BLOCK

// Device/Application/modbus/getObjIndexE
FUNCTION_BLOCK getObjIndexE
VAR_INPUT
	iI1:INT;
	iI2:INT;
END_VAR
VAR_OUTPUT
	iAdr:USINT;
END_VAR
VAR
	
END_VAR

//Modbus中，输入油缸编号索引，返回用于地址用于写入伸出状态是否到位
CASE iI1 OF
	1:
		CASE iI2 OF
			1:iAdr:=156;//L28
			2:iAdr:=157;//L29-L30
			3:iAdr:=126;	//L00
			4:iAdr:=119;		//Q29-Q30
			5:iAdr:=118;		//Q28
			6:iAdr:=142;//L01
		END_CASE
	2:
		CASE iI2 OF
			1:iAdr:=143;//L02-04
			2:iAdr:=144;//L05
			3:iAdr:=145;//L06-08
			4:iAdr:=146;//L09
			5:iAdr:=147;//L10-12
		END_CASE
	3:iAdr:=111;				//Q01-04
	4:iAdr:=112;				//Q05-08
	5:iAdr:=113;				//Q09-12
	6:
		CASE iI2 OF
			1:iAdr:=114;		//Q13-14
			2:iAdr:=115;		//Q15
			3:iAdr:=149;//L14-15
			4:iAdr:=148;//L13
			5:iAdr:=150;//L16
		END_CASE
	7:
		CASE iI2 OF
			1:iAdr:=152;//L18-21
			2:iAdr:=153;//L22
			3:iAdr:=154;//L23-26
			4:iAdr:=116;		//Q17-21
			5:iAdr:=117;		//Q22-26
			6:iAdr:=151;//L17
			7:iAdr:=155;//L27
		END_CASE

ELSE	
	iAdr:=0;
END_CASE

END_FUNCTION_BLOCK

// Device/Application/modbus/getObjIndexR
FUNCTION_BLOCK getObjIndexR
VAR_INPUT
	iI1:INT;
	iI2:INT;
END_VAR
VAR_OUTPUT
	iAdr:USINT;
END_VAR
VAR
	
END_VAR

//Modbus中，输入油缸编号索引，返回用于地址用于写入缩回状态是否到位
CASE iI1 OF
	1:		
		CASE iI2 OF	
			1:iAdr:=204;//L28
			2:iAdr:=205;//L29-30
			3:iAdr:=174;	//L00
			4:iAdr:=167;		//Q29-30
			5:iAdr:=166;		//Q28
			6:iAdr:=190;//L01
		END_CASE	
	2:		
		CASE iI2 OF	
			1:iAdr:=191;//L02-04
			2:iAdr:=192;//L05
			3:iAdr:=193;//L06-08
			4:iAdr:=194;//L09
			5:iAdr:=195;//L10-12
		END_CASE	
	3:iAdr:=159;				//Q01-04		
	4:iAdr:=160;				//Q05-08		
	5:iAdr:=161;				//Q09-12		
	6:		
		CASE iI2 OF	
			1:iAdr:=162;		//Q13-14
			2:iAdr:=163;		//Q15
			3:iAdr:=197;//L14-15
			4:iAdr:=196;//L13
			5:iAdr:=198;//L16
		END_CASE	
	7:		
		CASE iI2 OF	
			1:iAdr:=200;//L18-21
			2:iAdr:=201;//L22
			3:iAdr:=202;//L23-26
			4:iAdr:=164;		//Q17-21
			5:iAdr:=165;		//Q22-26
			6:iAdr:=199;//L17
			7:iAdr:=203;//L27
		END_CASE	


ELSE	
	iAdr:=0;
END_CASE

END_FUNCTION_BLOCK

// Device/Application/can/canRx
PROGRAM canRx
VAR
		T_CNT   :UINT;
END_VAR

T_CNT := T_CNT+1;
IF  T_CNT > 1000 THEN
	 T_CNT := 1;
END_IF


swmc_C05_Rx(T_CNT, ADR(gImple.PV_GroupTi));
swmc_C06_Rx(T_CNT, ADR(gImple.PV_GroupTi));
swmc_C12_Rx(T_CNT, ADR(gImple.PV_GroupTi));

END_PROGRAM

// Device/Application/can/swmc_C05_Rx
FUNCTION swmc_C05_Rx : BOOL
VAR_INPUT
	CNT				: UINT;

	psPVTi			: POINTER TO propValveModule_Ti;

END_VAR
VAR
	frame	 	    : Can_baseframe;
	COB_ID			: UINT;
	I				: UINT;
	Pre				: UINT;
	pos				: WORD;
END_VAR

IF gCan.C5RxMsg.RxCounter <>  gCan.C5RxCounter THEN    //接收到新的数据

	FOR  I := 1 TO  gCan.C5RxMsg.NoOfRxMessages DO
		frame :=CAN_Read_Data_SWMC(5,I);
		COB_ID :=	frame.id;    //获取ID
		CASE COB_ID OF     //根据ID解析协议
		
		//C5-0x350
			16#350://接收C5送来的数据
				pos := BYTE_TO_WORD(frame.data[1]) OR SHL(BYTE_TO_WORD(frame.data[2]),8);  	
				psPVTi^.arrPV[3].sNum[1].posVal.Current:= pos*0.1;
				pos := BYTE_TO_WORD(frame.data[3]) OR SHL(BYTE_TO_WORD(frame.data[4]),8);  
				psPVTi^.arrPV[3].sNum[2].posVal.Current:= pos*0.1;	
				pos := BYTE_TO_WORD(frame.data[5]) OR SHL(BYTE_TO_WORD(frame.data[6]),8);  
				psPVTi^.arrPV[3].sNum[3].posVal.Current:= pos*0.1;	
				pos := BYTE_TO_WORD(frame.data[7]) OR SHL(BYTE_TO_WORD(frame.data[8]),8);  	
				psPVTi^.arrPV[3].sNum[4].posVal.Current:= pos*0.1;
			
			//C5-0x351
			16#351://接收C5送来的数据
				pos := BYTE_TO_WORD(frame.data[1]) OR SHL(BYTE_TO_WORD(frame.data[2]),8);  	
				psPVTi^.arrPV[3].sNum[5].posVal.Current:= pos*0.1;	
				pos := BYTE_TO_WORD(frame.data[3]) OR SHL(BYTE_TO_WORD(frame.data[4]),8);  	
				psPVTi^.arrPV[3].sNum[6].posVal.Current:= pos*0.1;	
				pos := BYTE_TO_WORD(frame.data[5]) OR SHL(BYTE_TO_WORD(frame.data[6]),8);  	
				psPVTi^.arrPV[3].sNum[7].posVal.Current:= pos*0.1;	
				pos := BYTE_TO_WORD(frame.data[7]) OR SHL(BYTE_TO_WORD(frame.data[8]),8);  	
				psPVTi^.arrPV[3].sNum[8].posVal.Current:= pos*0.1;
			
			//C5-0x352
			16#352://接收C5送来的数据
			pos := BYTE_TO_WORD(frame.data[1]) OR SHL(BYTE_TO_WORD(frame.data[2]),8);  	
				psPVTi^.arrPV[4].sNum[1].posVal.Current:= pos*0.1;	
				pos := BYTE_TO_WORD(frame.data[3]) OR SHL(BYTE_TO_WORD(frame.data[4]),8);  	
				psPVTi^.arrPV[4].sNum[2].posVal.Current:= pos*0.1;		
				pos := BYTE_TO_WORD(frame.data[5]) OR SHL(BYTE_TO_WORD(frame.data[6]),8);  	
				psPVTi^.arrPV[4].sNum[3].posVal.Current:= pos*0.1;		
				pos := BYTE_TO_WORD(frame.data[7]) OR SHL(BYTE_TO_WORD(frame.data[8]),8);  	
				psPVTi^.arrPV[4].sNum[4].posVal.Current:= pos*0.1;	
			
			//C5-0x353
			16#353://接收C5送来的数据
				pos := BYTE_TO_WORD(frame.data[1]) OR SHL(BYTE_TO_WORD(frame.data[2]),8);  	
				psPVTi^.arrPV[4].sNum[5].posVal.Current:= pos*0.1;		
				pos := BYTE_TO_WORD(frame.data[3]) OR SHL(BYTE_TO_WORD(frame.data[4]),8);  	
				psPVTi^.arrPV[4].sNum[6].posVal.Current:= pos*0.1;		
				pos := BYTE_TO_WORD(frame.data[5]) OR SHL(BYTE_TO_WORD(frame.data[6]),8);  	
				psPVTi^.arrPV[4].sNum[7].posVal.Current:= pos*0.1;		
				pos := BYTE_TO_WORD(frame.data[7]) OR SHL(BYTE_TO_WORD(frame.data[8]),8);  	
				psPVTi^.arrPV[4].sNum[8].posVal.Current:= pos*0.1;	
			
			//C5-0x354
			16#354://接收C5送来的数据
			pos := BYTE_TO_WORD(frame.data[1]) OR SHL(BYTE_TO_WORD(frame.data[2]),8);  	
				psPVTi^.arrPV[5].sNum[1].posVal.Current:= pos*0.1;		
				pos := BYTE_TO_WORD(frame.data[3]) OR SHL(BYTE_TO_WORD(frame.data[4]),8);  	
				psPVTi^.arrPV[5].sNum[2].posVal.Current:= pos*0.1;		
				pos := BYTE_TO_WORD(frame.data[5]) OR SHL(BYTE_TO_WORD(frame.data[6]),8);  	
				psPVTi^.arrPV[5].sNum[3].posVal.Current:= pos*0.1;		
				pos := BYTE_TO_WORD(frame.data[7]) OR SHL(BYTE_TO_WORD(frame.data[8]),8);  	
				psPVTi^.arrPV[5].sNum[4].posVal.Current:= pos*0.1;	
			
			//C5-0x355
			16#355://接收C5送来的数据
			pos := BYTE_TO_WORD(frame.data[1]) OR SHL(BYTE_TO_WORD(frame.data[2]),8);  	
				psPVTi^.arrPV[5].sNum[5].posVal.Current:= pos*0.1;		
				pos := BYTE_TO_WORD(frame.data[3]) OR SHL(BYTE_TO_WORD(frame.data[4]),8);  	
				psPVTi^.arrPV[5].sNum[6].posVal.Current:= pos*0.1;		
				pos := BYTE_TO_WORD(frame.data[5]) OR SHL(BYTE_TO_WORD(frame.data[6]),8);  	
				psPVTi^.arrPV[5].sNum[7].posVal.Current:= pos*0.1;		
				pos := BYTE_TO_WORD(frame.data[7]) OR SHL(BYTE_TO_WORD(frame.data[8]),8);  	
				psPVTi^.arrPV[5].sNum[8].posVal.Current:= pos*0.1;	
			

	
			//C5-0x356
			16#356:           //接收C5送来的数据
			(*
				Pre :=BYTE_TO_WORD(frame.data[1]) OR SHL(BYTE_TO_WORD(frame.data[2]),8);
				psYyz^.Status.pressureV10:= 	(Pre-4000)/16000.0*400;	
				Pre :=BYTE_TO_WORD(frame.data[3]) OR SHL(BYTE_TO_WORD(frame.data[4]),8);
				psYyz^.Status.pressureV11:= 	(Pre-4000)/16000.0*400;	
			*)
			
	
		END_CASE
	END_FOR
	gCan.C5RxCounter := gCan.C5RxMsg.RxCounter ;
END_IF

END_FUNCTION

// Device/Application/can/CAN_Read_Data_SWMC
FUNCTION CAN_Read_Data_SWMC : Can_baseframe
VAR_INPUT
	SWMC_ID	 :UINT;		//接收SWMC控制ID
	I	 	 :UINT;      //接收缓冲区域
END_VAR
VAR
	frame :Can_baseframe;
END_VAR

CASE  SWMC_ID OF

	5:                       //SWMC-C5
		frame.id 	:= (gCan.C5RxMsg.RXMsg[I].RxMsg_CobId-8)/32;
		frame.data 	:= gCan.C5RxMsg.RXMsg[I].RxMsg_Byte;
				
	6:                       //SWMC-C6
		frame.id 	:= (gCan.C6RxMsg.RXMsg[I].RxMsg_CobId-8)/32;
		frame.data 	:= gCan.C6RxMsg.RXMsg[I].RxMsg_Byte;

	12:						//SWMC-C12
		frame.id 	:= (gCan.C12RxMsg.RXMsg[I].RxMsg_CobId-8)/32;
		frame.data 	:= gCan.C12RxMsg.RXMsg[I].RxMsg_Byte;	
		
	ELSE				//Other
		frame.id := 0;
		frame.data[1] := 0;
		frame.data[2] := 0;
		frame.data[3] := 0;
		frame.data[4] := 0;
		frame.data[5] := 0;
		frame.data[6] := 0;
		frame.data[7] := 0;
		frame.data[8] := 0;
END_CASE
Can_Read_data_SWMC := frame;

END_FUNCTION

// Device/Application/can/swmc_C06_Rx
FUNCTION swmc_C06_Rx : BOOL
VAR_INPUT
	CNT				: UINT;

	psPVTi			: POINTER TO propValveModule_Ti;

END_VAR
VAR
	frame	 	    : Can_baseframe;
	COB_ID			: UINT;
	I				: UINT;
	Pre				: UINT;
	pos				: WORD;
END_VAR

IF gCan.C6RxMsg.RxCounter <>  gCan.C6RxCounter THEN    //接收到新的数据

	FOR  I := 1 TO  gCan.C6RxMsg.NoOfRxMessages DO
		frame :=CAN_Read_Data_SWMC(6,I);
		COB_ID :=	frame.id;    //获取ID
		CASE COB_ID OF     //根据ID解析协议
	
		
			//C6-0x360
			16#360:           //接收C6送来的数据
				pos:=BYTE_TO_WORD(frame.data[1]) OR SHL(BYTE_TO_WORD(frame.data[2]),8);
				psPVTi^.arrPV[1].sNum[3].posVal.Current:=pos*0.1;
				pos:=BYTE_TO_WORD(frame.data[3]) OR SHL(BYTE_TO_WORD(frame.data[4]),8);
				psPVTi^.arrPV[1].sNum[4].posVal.Current:=pos*0.1;
				pos:=BYTE_TO_WORD(frame.data[5]) OR SHL(BYTE_TO_WORD(frame.data[6]),8);
				psPVTi^.arrPV[1].sNum[9].posVal.Current:=pos*0.1;
				pos:=BYTE_TO_WORD(frame.data[7]) OR SHL(BYTE_TO_WORD(frame.data[8]),8);
				psPVTi^.arrPV[1].sNum[5].posVal.Current:=pos*0.1;
			

			//C6-0x361
			16#361:           //接收C6送来的数据
				pos:=BYTE_TO_WORD(frame.data[1]) OR SHL(BYTE_TO_WORD(frame.data[2]),8);
				psPVTi^.arrPV[1].sNum[8].posVal.Current:=pos*0.1;
				pos:=BYTE_TO_WORD(frame.data[3]) OR SHL(BYTE_TO_WORD(frame.data[4]),8);
				psPVTi^.arrPV[1].sNum[6].posVal.Current:=pos*0.1;
				pos:=BYTE_TO_WORD(frame.data[5]) OR SHL(BYTE_TO_WORD(frame.data[6]),8);
				psPVTi^.arrPV[1].sNum[7].posVal.Current:=pos*0.1;
				pos:=BYTE_TO_WORD(frame.data[7]) OR SHL(BYTE_TO_WORD(frame.data[8]),8);
				psPVTi^.arrPV[2].sNum[1].posVal.Current:=pos*0.1;
			//C6-0x362
			16#362:           //接收C6送来的数据
				pos:=BYTE_TO_WORD(frame.data[1]) OR SHL(BYTE_TO_WORD(frame.data[2]),8);
				psPVTi^.arrPV[2].sNum[2].posVal.Current:=pos*0.1;
				pos:=BYTE_TO_WORD(frame.data[3]) OR SHL(BYTE_TO_WORD(frame.data[4]),8);
				psPVTi^.arrPV[2].sNum[3].posVal.Current:=pos*0.1;
				pos:=BYTE_TO_WORD(frame.data[5]) OR SHL(BYTE_TO_WORD(frame.data[6]),8);
				psPVTi^.arrPV[2].sNum[4].posVal.Current:=pos*0.1;
				pos:=BYTE_TO_WORD(frame.data[7]) OR SHL(BYTE_TO_WORD(frame.data[8]),8);
				psPVTi^.arrPV[2].sNum[5].posVal.Current:=pos*0.1;
			//C6-0x363
			16#363:           //接收C6送来的数据
				pos:=BYTE_TO_WORD(frame.data[1]) OR SHL(BYTE_TO_WORD(frame.data[2]),8);
				psPVTi^.arrPV[2].sNum[6].posVal.Current:=pos*0.1;
				pos:=BYTE_TO_WORD(frame.data[3]) OR SHL(BYTE_TO_WORD(frame.data[4]),8);
				psPVTi^.arrPV[2].sNum[7].posVal.Current:=pos*0.1;
				pos:=BYTE_TO_WORD(frame.data[5]) OR SHL(BYTE_TO_WORD(frame.data[6]),8);
				psPVTi^.arrPV[2].sNum[8].posVal.Current:=pos*0.1;
				pos:=BYTE_TO_WORD(frame.data[7]) OR SHL(BYTE_TO_WORD(frame.data[8]),8);
				psPVTi^.arrPV[2].sNum[9].posVal.Current:=pos*0.1;
			//C6-0x364
			16#364:           //接收C6送来的数据
				pos:=BYTE_TO_WORD(frame.data[1]) OR SHL(BYTE_TO_WORD(frame.data[2]),8);
				psPVTi^.arrPV[2].sNum[10].posVal.Current:=pos*0.1;
				pos:=BYTE_TO_WORD(frame.data[3]) OR SHL(BYTE_TO_WORD(frame.data[4]),8);
				psPVTi^.arrPV[2].sNum[11].posVal.Current:=pos*0.1;
				pos:=BYTE_TO_WORD(frame.data[5]) OR SHL(BYTE_TO_WORD(frame.data[6]),8);
				psPVTi^.arrPV[6].sNum[6].posVal.Current:=pos*0.1;
				pos:=BYTE_TO_WORD(frame.data[7]) OR SHL(BYTE_TO_WORD(frame.data[8]),8);
				psPVTi^.arrPV[6].sNum[4].posVal.Current:=pos*0.1;
			//C6-0x365
			16#365:           //接收C6送来的数据
				pos:=BYTE_TO_WORD(frame.data[1]) OR SHL(BYTE_TO_WORD(frame.data[2]),8);
				psPVTi^.arrPV[6].sNum[5].posVal.Current:=pos*0.1;
				pos:=BYTE_TO_WORD(frame.data[3]) OR SHL(BYTE_TO_WORD(frame.data[4]),8);
				psPVTi^.arrPV[6].sNum[1].posVal.Current:=pos*0.1;
				pos:=BYTE_TO_WORD(frame.data[5]) OR SHL(BYTE_TO_WORD(frame.data[6]),8);
				psPVTi^.arrPV[6].sNum[2].posVal.Current:=pos*0.1;
				pos:=BYTE_TO_WORD(frame.data[7]) OR SHL(BYTE_TO_WORD(frame.data[8]),8);
				psPVTi^.arrPV[6].sNum[3].posVal.Current:=pos*0.1;
				
		
